LIN {X 0,Y 418.25,Z 362.008,A -85,B 0,C 180,E1 -10239.337,E2 -10239.337} C_VEL
LIN {X 0,Y 418.278,Z 362.011,A -85,B 0,C 180,E1 -10242.396,E2 -10242.396} C_VEL
LIN {X 0,Y 418.299,Z 362.002,A -85,B 0,C 180,E1 -10245.403,E2 -10245.403} C_VEL
LIN {X 0,Y 418.315,Z 361.999,A -85,B 0,C 180,E1 -10248.369,E2 -10248.369} C_VEL
LIN {X 0,Y 418.378,Z 361.987,A -85,B 0,C 180,E1 -10251.305,E2 -10251.305} C_VEL
LIN {X 0,Y 418.49,Z 361.983,A -85,B 0,C 180,E1 -10254.217,E2 -10254.217} C_VEL
LIN {X 0,Y 418.542,Z 361.975,A -85,B 0,C 180,E1 -10258.076,E2 -10258.076} C_VEL
LIN {X 0,Y 418.475,Z 361.982,A -85,B 0,C 180,E1 -10260.963,E2 -10260.963} C_VEL
LIN {X 0,Y 418.488,Z 361.975,A -85,B 0,C 180,E1 -10262.888,E2 -10262.888} C_VEL
LIN {X 0,Y 418.445,Z 361.981,A -85,B 0,C 180,E1 -10266.567,E2 -10266.567} C_VEL
LIN {X 0,Y 418.34,Z 361.998,A -85,B 0,C 180,E1 -10269.672,E2 -10269.672} C_VEL
LIN {X 0,Y 418.349,Z 361.997,A -85,B 0,C 180,E1 -10273.001,E2 -10273.001} C_VEL
LIN {X 0,Y 418.315,Z 362.003,A -85,B 0,C 180,E1 -10276.736,E2 -10276.736} C_VEL
LIN {X 0,Y 418.273,Z 361.985,A -85,B 0,C 180,E1 -10279.79,E2 -10279.79} C_VEL
LIN {X 0,Y 418.233,Z 362.015,A -85,B 0,C 180,E1 -10282.737,E2 -10282.737} C_VEL
LIN {X 0,Y 418.233,Z 361.994,A -85,B 0,C 180,E1 -10285.907,E2 -10285.907} C_VEL
LIN {X 0,Y 418.263,Z 362.006,A -85,B 0,C 180,E1 -10289.163,E2 -10289.163} C_VEL
LIN {X 0,Y 418.26,Z 362.012,A -85,B 0,C 180,E1 -10292.844,E2 -10292.844} C_VEL
LIN {X 0,Y 418.244,Z 362.002,A -85,B 0,C 180,E1 -10296.237,E2 -10296.237} C_VEL
LIN {X 0,Y 418.201,Z 362.009,A -85,B 0,C 180,E1 -10299.688,E2 -10299.688} C_VEL
LIN {X 0,Y 418.215,Z 362.01,A -85,B 0,C 180,E1 -10302.319,E2 -10302.319} C_VEL
LIN {X 0,Y 418.239,Z 362.007,A -85,B 0,C 180,E1 -10305.109,E2 -10305.109} C_VEL
LIN {X 0,Y 418.238,Z 362.008,A -85,B 0,C 180,E1 -10307.766,E2 -10307.766} C_VEL
LIN {X 0,Y 418.259,Z 362.142,A -85,B 0,C 180,E1 -10309.979,E2 -10309.979} C_VEL
LIN {X 0,Y 420.964,Z 372.598,A -85,B 0,C 180,E1 -10312.371,E2 -10312.371} C_VEL
LIN {X 0,Y 430.235,Z 392.629,A -85,B 0,C 180,E1 -10313.476,E2 -10313.476} C_VEL
LIN {X 0,Y 432.008,Z 399.713,A -85,B 0,C 180,E1 -10313.741,E2 -10313.741} C_VEL
LIN {X 0,Y 429.477,Z 524.303,A -85,B 0,C 180,E1 -10315.876,E2 -10315.876} C_VEL
LIN {X 0,Y 429.158,Z 541.846,A -85,B 0,C 180,E1 -10316.252,E2 -10316.252} C_VEL
LIN {X 0,Y 428.401,Z 556.662,A -85,B 0,C 180,E1 -10316.74,E2 -10316.74} C_VEL
LIN {X 0,Y 427.518,Z 571.385,A -85,B 0,C 180,E1 -10317.427,E2 -10317.427} C_VEL
LIN {X 0,Y 426.537,Z 583.995,A -85,B 0,C 180,E1 -10318.179,E2 -10318.179} C_VEL
LIN {X 0,Y 425.351,Z 597.555,A -85,B 0,C 180,E1 -10319.189,E2 -10319.189} C_VEL
LIN {X 0,Y 424.073,Z 610.048,A -85,B 0,C 180,E1 -10320.323,E2 -10320.323} C_VEL
LIN {X 0,Y 422.821,Z 621.605,A -85,B 0,C 180,E1 -10321.586,E2 -10321.586} C_VEL
LIN {X 0,Y 421.617,Z 632.292,A -85,B 0,C 180,E1 -10322.984,E2 -10322.984} C_VEL
LIN {X 0,Y 420.39,Z 642.896,A -85,B 0,C 180,E1 -10324.64,E2 -10324.64} C_VEL
LIN {X 0,Y 419.394,Z 651.646,A -85,B 0,C 180,E1 -10326.285,E2 -10326.285} C_VEL
LIN {X 0,Y 418.644,Z 659.535,A -85,B 0,C 180,E1 -10328.074,E2 -10328.074} C_VEL
LIN {X 0,Y 417.946,Z 665.94,A -85,B 0,C 180,E1 -10329.835,E2 -10329.835} C_VEL
LIN {X 0,Y 417.521,Z 671.781,A -85,B 0,C 180,E1 -10331.856,E2 -10331.856} C_VEL
LIN {X 0,Y 417.395,Z 673.436,A -85,B 0,C 180,E1 -10332.537,E2 -10332.537} C_VEL
LIN {X 0,Y 416.6,Z 675.164,A -85,B 0,C 180,E1 -10333.308,E2 -10333.308} C_VEL
LIN {X 0,Y 413.563,Z 677.628,A -85,B 0,C 180,E1 -10334.568,E2 -10334.568} C_VEL
LIN {X 0,Y 411.054,Z 679.223,A -85,B 0,C 180,E1 -10335.596,E2 -10335.596} C_VEL
LIN {X 0,Y 409.922,Z 680.326,A -85,B 0,C 180,E1 -10336.536,E2 -10336.536} C_VEL
LIN {X 0,Y 409.899,Z 680.381,A -85,B 0,C 180,E1 -10336.673,E2 -10336.673} C_VEL
LIN {X 0,Y 409.94,Z 681.451,A -85,B 0,C 180,E1 -10338.128,E2 -10338.128} C_VEL
LIN {X 0,Y 409.796,Z 681.883,A -85,B 0,C 180,E1 -10340.125,E2 -10340.125} C_VEL
LIN {X 0,Y 409.865,Z 681.164,A -85,B 0,C 180,E1 -10342.116,E2 -10342.116} C_VEL
LIN {X 0,Y 410.059,Z 679.25,A -85,B 0,C 180,E1 -10344.098,E2 -10344.098} C_VEL
LIN {X 0,Y 410.126,Z 676.158,A -85,B 0,C 180,E1 -10346.07,E2 -10346.07} C_VEL
LIN {X 0,Y 410.35,Z 671.836,A -85,B 0,C 180,E1 -10348.037,E2 -10348.037} C_VEL
LIN {X 0,Y 410.68,Z 666.199,A -85,B 0,C 180,E1 -10350,E2 -10350} C_VEL
LIN {X 0,Y 411.345,Z 659.076,A -85,B 0,C 180,E1 -10351.958,E2 -10351.958} C_VEL
LIN {X 0,Y 412.106,Z 651.471,A -85,B 0,C 180,E1 -10353.667,E2 -10353.667} C_VEL
LIN {X 0,Y 413.018,Z 642.359,A -85,B 0,C 180,E1 -10355.37,E2 -10355.37} C_VEL
LIN {X 0,Y 414.008,Z 633.119,A -85,B 0,C 180,E1 -10356.825,E2 -10356.825} C_VEL
LIN {X 0,Y 415.304,Z 621.14,A -85,B 0,C 180,E1 -10358.393,E2 -10358.393} C_VEL
LIN {X 0,Y 416.452,Z 608.984,A -85,B 0,C 180,E1 -10359.716,E2 -10359.716} C_VEL
LIN {X 0,Y 417.684,Z 595.584,A -85,B 0,C 180,E1 -10360.912,E2 -10360.912} C_VEL
LIN {X 0,Y 418.769,Z 582.449,A -85,B 0,C 180,E1 -10361.864,E2 -10361.864} C_VEL
LIN {X 0,Y 419.759,Z 568,A -85,B 0,C 180,E1 -10362.695,E2 -10362.695} C_VEL
LIN {X 0,Y 420.566,Z 552.989,A -85,B 0,C 180,E1 -10363.345,E2 -10363.345} C_VEL
LIN {X 0,Y 421.105,Z 537.257,A -85,B 0,C 180,E1 -10363.82,E2 -10363.82} C_VEL
LIN {X 0,Y 423.525,Z 401.204,A -85,B 0,C 180,E1 -10366.178,E2 -10366.178} C_VEL
LIN {X 0,Y 422.464,Z 395.65,A -85,B 0,C 180,E1 -10366.343,E2 -10366.343} C_VEL
LIN {X 0,Y 421.07,Z 390.956,A -85,B 0,C 180,E1 -10366.513,E2 -10366.513} C_VEL
LIN {X 0,Y 413.404,Z 372.221,A -85,B 0,C 180,E1 -10367.36,E2 -10367.36} C_VEL
LIN {X 0,Y 411.282,Z 362.882,A -85,B 0,C 180,E1 -10369.399,E2 -10369.399} C_VEL
LIN {X 0,Y 411.194,Z 362.89,A -85,B 0,C 180,E1 -10373.148,E2 -10373.148} C_VEL
LIN {X 0,Y 411.18,Z 362.89,A -85,B 0,C 180,E1 -10376.385,E2 -10376.385} C_VEL
LIN {X 0,Y 411.201,Z 362.886,A -85,B 0,C 180,E1 -10379.713,E2 -10379.713} C_VEL
LIN {X 0,Y 411.211,Z 362.881,A -85,B 0,C 180,E1 -10383.156,E2 -10383.156} C_VEL
LIN {X 0,Y 411.193,Z 362.881,A -85,B 0,C 180,E1 -10386.552,E2 -10386.552} C_VEL
LIN {X 0,Y 411.171,Z 362.886,A -85,B 0,C 180,E1 -10389.72,E2 -10389.72} C_VEL
LIN {X 0,Y 411.166,Z 362.892,A -85,B 0,C 180,E1 -10393.135,E2 -10393.135} C_VEL
LIN {X 0,Y 411.169,Z 362.881,A -85,B 0,C 180,E1 -10395.881,E2 -10395.881} C_VEL
LIN {X 0,Y 411.152,Z 362.892,A -85,B 0,C 180,E1 -10398.774,E2 -10398.774} C_VEL
LIN {X 0,Y 411.186,Z 362.89,A -85,B 0,C 180,E1 -10402.025,E2 -10402.025} C_VEL
LIN {X 0,Y 411.206,Z 362.887,A -85,B 0,C 180,E1 -10405.123,E2 -10405.123} C_VEL
LIN {X 0,Y 411.167,Z 362.894,A -85,B 0,C 180,E1 -10408.002,E2 -10408.002} C_VEL
LIN {X 0,Y 411.179,Z 362.878,A -85,B 0,C 180,E1 -10411.406,E2 -10411.406} C_VEL
LIN {X 0,Y 411.191,Z 362.861,A -85,B 0,C 180,E1 -10414.941,E2 -10414.941} C_VEL
LIN {X 0,Y 411.207,Z 362.888,A -85,B 0,C 180,E1 -10417.913,E2 -10417.913} C_VEL
LIN {X 0,Y 411.223,Z 362.883,A -85,B 0,C 180,E1 -10421.051,E2 -10421.051} C_VEL
LIN {X 0,Y 411.257,Z 362.879,A -85,B 0,C 180,E1 -10424.131,E2 -10424.131} C_VEL
LIN {X 0,Y 411.307,Z 362.873,A -85,B 0,C 180,E1 -10427.165,E2 -10427.165} C_VEL
LIN {X 0,Y 411.291,Z 362.873,A -85,B 0,C 180,E1 -10430.161,E2 -10430.161} C_VEL
LIN {X 0,Y 411.393,Z 362.862,A -85,B 0,C 180,E1 -10433.131,E2 -10433.131} C_VEL
LIN {X 0,Y 411.291,Z 362.866,A -85,B 0,C 180,E1 -10435.098,E2 -10435.098} C_VEL
LIN {X 0,Y 411.505,Z 362.849,A -85,B 0,C 180,E1 -10438.042,E2 -10438.042} C_VEL
LIN {X 0,Y 411.517,Z 362.843,A -85,B 0,C 180,E1 -10440,E2 -10440} C_VEL
LIN {X 0,Y 411.449,Z 362.85,A -85,B 0,C 180,E1 -10442.937,E2 -10442.937} C_VEL
LIN {X 0,Y 411.432,Z 362.858,A -85,B 0,C 180,E1 -10445.882,E2 -10445.882} C_VEL
LIN {X 0,Y 411.32,Z 362.866,A -85,B 0,C 180,E1 -10448.846,E2 -10448.846} C_VEL
LIN {X 0,Y 411.285,Z 362.873,A -85,B 0,C 180,E1 -10451.832,E2 -10451.832} C_VEL
LIN {X 0,Y 411.233,Z 362.879,A -85,B 0,C 180,E1 -10454.853,E2 -10454.853} C_VEL
LIN {X 0,Y 411.231,Z 362.878,A -85,B 0,C 180,E1 -10457.916,E2 -10457.916} C_VEL
LIN {X 0,Y 411.198,Z 362.885,A -85,B 0,C 180,E1 -10461.034,E2 -10461.034} C_VEL
LIN {X 0,Y 411.204,Z 362.886,A -85,B 0,C 180,E1 -10464.216,E2 -10464.216} C_VEL
LIN {X 0,Y 411.176,Z 362.891,A -85,B 0,C 180,E1 -10467.483,E2 -10467.483} C_VEL
LIN {X 0,Y 411.197,Z 362.888,A -85,B 0,C 180,E1 -10469.713,E2 -10469.713} C_VEL
LIN {X 0,Y 411.207,Z 362.886,A -85,B 0,C 180,E1 -10473.155,E2 -10473.155} C_VEL
LIN {X 0,Y 411.189,Z 362.887,A -85,B 0,C 180,E1 -10476.551,E2 -10476.551} C_VEL
LIN {X 0,Y 411.167,Z 362.886,A -85,B 0,C 180,E1 -10479.72,E2 -10479.72} C_VEL
LIN {X 0,Y 411.162,Z 362.892,A -85,B 0,C 180,E1 -10483.135,E2 -10483.135} C_VEL
LIN {X 0,Y 411.164,Z 362.895,A -85,B 0,C 180,E1 -10485.881,E2 -10485.881} C_VEL
LIN {X 0,Y 411.148,Z 362.896,A -85,B 0,C 180,E1 -10488.774,E2 -10488.774} C_VEL
LIN {X 0,Y 411.182,Z 362.891,A -85,B 0,C 180,E1 -10492.025,E2 -10492.025} C_VEL
LIN {X 0,Y 411.204,Z 362.891,A -85,B 0,C 180,E1 -10495.666,E2 -10495.666} C_VEL
LIN {X 0,Y 411.212,Z 362.956,A -85,B 0,C 180,E1 -10497.008,E2 -10497.008} C_VEL
LIN {X 0,Y 414.98,Z 378.406,A -85,B 0,C 180,E1 -10500.005,E2 -10500.005} C_VEL
LIN {X 0,Y 417.196,Z 388.376,A -85,B 0,C 180,E1 -10501.856,E2 -10501.856} C_VEL
LIN {X 0,Y 416.892,Z 394.781,A -85,B 0,C 180,E1 -10502.901,E2 -10502.901} C_VEL
LIN {X 0,Y 423.237,Z 429.477,A -85,B 0,C 180,E1 -10503.921,E2 -10503.921} C_VEL
LIN {X 0,Y 420.919,Z 561.659,A -85,B 0,C 180,E1 -10506.213,E2 -10506.213} C_VEL
LIN {X 0,Y 420.155,Z 577.601,A -85,B 0,C 180,E1 -10506.689,E2 -10506.689} C_VEL
LIN {X 0,Y 419.305,Z 592.288,A -85,B 0,C 180,E1 -10507.325,E2 -10507.325} C_VEL
LIN {X 0,Y 418.178,Z 607.066,A -85,B 0,C 180,E1 -10508.171,E2 -10508.171} C_VEL
LIN {X 0,Y 417.022,Z 620.494,A -85,B 0,C 180,E1 -10509.144,E2 -10509.144} C_VEL
LIN {X 0,Y 415.674,Z 634.123,A -85,B 0,C 180,E1 -10510.364,E2 -10510.364} C_VEL
LIN {X 0,Y 414.455,Z 646.627,A -85,B 0,C 180,E1 -10511.732,E2 -10511.732} C_VEL
LIN {X 0,Y 413.378,Z 657.812,A -85,B 0,C 180,E1 -10513.2,E2 -10513.2} C_VEL
LIN {X 0,Y 412.375,Z 667.299,A -85,B 0,C 180,E1 -10514.683,E2 -10514.683} C_VEL
LIN {X 0,Y 411.614,Z 675.377,A -85,B 0,C 180,E1 -10516.17,E2 -10516.17} C_VEL
LIN {X 0,Y 410.988,Z 683.35,A -85,B 0,C 180,E1 -10517.908,E2 -10517.908} C_VEL
LIN {X 0,Y 410.506,Z 689.961,A -85,B 0,C 180,E1 -10519.644,E2 -10519.644} C_VEL
LIN {X 0,Y 410.206,Z 696.028,A -85,B 0,C 180,E1 -10521.626,E2 -10521.626} C_VEL
LIN {X 0,Y 410.056,Z 699.608,A -85,B 0,C 180,E1 -10523.109,E2 -10523.109} C_VEL
LIN {X 0,Y 409.958,Z 703.281,A -85,B 0,C 180,E1 -10525.083,E2 -10525.083} C_VEL
LIN {X 0,Y 409.919,Z 705.726,A -85,B 0,C 180,E1 -10527.052,E2 -10527.052} C_VEL
LIN {X 0,Y 409.935,Z 706.987,A -85,B 0,C 180,E1 -10529.018,E2 -10529.018} C_VEL
LIN {X 0,Y 409.935,Z 707.048,A -85,B 0,C 180,E1 -10530.982,E2 -10530.982} C_VEL
LIN {X 0,Y 409.916,Z 705.971,A -85,B 0,C 180,E1 -10532.948,E2 -10532.948} C_VEL
LIN {X 0,Y 409.94,Z 703.747,A -85,B 0,C 180,E1 -10534.917,E2 -10534.917} C_VEL
LIN {X 0,Y 410.048,Z 700.335,A -85,B 0,C 180,E1 -10536.891,E2 -10536.891} C_VEL
LIN {X 0,Y 410.274,Z 695.646,A -85,B 0,C 180,E1 -10538.869,E2 -10538.869} C_VEL
LIN {X 0,Y 410.686,Z 689.548,A -85,B 0,C 180,E1 -10540.85,E2 -10540.85} C_VEL
LIN {X 0,Y 411.23,Z 682.928,A -85,B 0,C 180,E1 -10542.586,E2 -10542.586} C_VEL
LIN {X 0,Y 412.029,Z 675.001,A -85,B 0,C 180,E1 -10544.319,E2 -10544.319} C_VEL
LIN {X 0,Y 413.047,Z 665.51,A -85,B 0,C 180,E1 -10546.051,E2 -10546.051} C_VEL
LIN {X 0,Y 414.218,Z 655.864,A -85,B 0,C 180,E1 -10547.527,E2 -10547.527} C_VEL
LIN {X 0,Y 415.508,Z 644.448,A -85,B 0,C 180,E1 -10549.002,E2 -10549.002} C_VEL
LIN {X 0,Y 416.82,Z 633.191,A -85,B 0,C 180,E1 -10550.221,E2 -10550.221} C_VEL
LIN {X 0,Y 418.291,Z 619.612,A -85,B 0,C 180,E1 -10551.434,E2 -10551.434} C_VEL
LIN {X 0,Y 419.597,Z 606.311,A -85,B 0,C 180,E1 -10552.399,E2 -10552.399} C_VEL
LIN {X 0,Y 420.822,Z 591.552,A -85,B 0,C 180,E1 -10553.246,E2 -10553.246} C_VEL
LIN {X 0,Y 421.861,Z 576.455,A -85,B 0,C 180,E1 -10553.893,E2 -10553.893} C_VEL
LIN {X 0,Y 422.653,Z 561.479,A -85,B 0,C 180,E1 -10554.335,E2 -10554.335} C_VEL
LIN {X 0,Y 424.423,Z 477.264,A -85,B 0,C 180,E1 -10555.827,E2 -10555.827} C_VEL
LIN {X 0,Y 425.245,Z 428.739,A -85,B 0,C 180,E1 -10556.686,E2 -10556.686} C_VEL
LIN {X 0,Y 420.958,Z 406.331,A -85,B 0,C 180,E1 -10557.445,E2 -10557.445} C_VEL
LIN {X 0,Y 418.176,Z 394.198,A -85,B 0,C 180,E1 -10557.913,E2 -10557.913} C_VEL
LIN {X 0,Y 418.264,Z 390.82,A -85,B 0,C 180,E1 -10558.508,E2 -10558.508} C_VEL
LIN {X 0,Y 415.766,Z 379.592,A -85,B 0,C 180,E1 -10560.752,E2 -10560.752} C_VEL
LIN {X 0,Y 411.97,Z 365.752,A -85,B 0,C 180,E1 -10563.716,E2 -10563.716} C_VEL
LIN {X 0,Y 411.242,Z 362.886,A -85,B 0,C 180,E1 -10564.398,E2 -10564.398} C_VEL
LIN {X 0,Y 411.191,Z 362.888,A -85,B 0,C 180,E1 -10568.166,E2 -10568.166} C_VEL
LIN {X 0,Y 411.162,Z 362.885,A -85,B 0,C 180,E1 -10571.807,E2 -10571.807} C_VEL
LIN {X 0,Y 411.173,Z 362.892,A -85,B 0,C 180,E1 -10575.51,E2 -10575.51} C_VEL
LIN {X 0,Y 411.146,Z 362.897,A -85,B 0,C 180,E1 -10578.775,E2 -10578.775} C_VEL
LIN {X 0,Y 411.181,Z 362.892,A -85,B 0,C 180,E1 -10582.025,E2 -10582.025} C_VEL
LIN {X 0,Y 411.205,Z 362.883,A -85,B 0,C 180,E1 -10585.667,E2 -10585.667} C_VEL
LIN {X 0,Y 411.188,Z 362.868,A -85,B 0,C 180,E1 -10589.153,E2 -10589.153} C_VEL
LIN {X 0,Y 411.188,Z 362.89,A -85,B 0,C 180,E1 -10592.518,E2 -10592.518} C_VEL
LIN {X 0,Y 411.211,Z 362.886,A -85,B 0,C 180,E1 -10595.784,E2 -10595.784} C_VEL
LIN {X 0,Y 411.197,Z 362.888,A -85,B 0,C 180,E1 -10598.966,E2 -10598.966} C_VEL
LIN {X 0,Y 411.244,Z 362.883,A -85,B 0,C 180,E1 -10602.085,E2 -10602.085} C_VEL
LIN {X 0,Y 411.256,Z 362.88,A -85,B 0,C 180,E1 -10605.148,E2 -10605.148} C_VEL
LIN {X 0,Y 411.284,Z 362.873,A -85,B 0,C 180,E1 -10608.168,E2 -10608.168} C_VEL
LIN {X 0,Y 411.319,Z 362.867,A -85,B 0,C 180,E1 -10611.154,E2 -10611.154} C_VEL
LIN {X 0,Y 411.435,Z 362.861,A -85,B 0,C 180,E1 -10614.118,E2 -10614.118} C_VEL
LIN {X 0,Y 411.511,Z 362.851,A -85,B 0,C 180,E1 -10618.043,E2 -10618.043} C_VEL
LIN {X 0,Y 411.439,Z 362.859,A -85,B 0,C 180,E1 -10620.979,E2 -10620.979} C_VEL
LIN {X 0,Y 411.445,Z 362.851,A -85,B 0,C 180,E1 -10622.938,E2 -10622.938} C_VEL
LIN {X 0,Y 411.394,Z 362.858,A -85,B 0,C 180,E1 -10626.564,E2 -10626.564} C_VEL
LIN {X 0,Y 411.292,Z 362.876,A -85,B 0,C 180,E1 -10629.839,E2 -10629.839} C_VEL
LIN {X 0,Y 411.308,Z 362.874,A -85,B 0,C 180,E1 -10633.105,E2 -10633.105} C_VEL
LIN {X 0,Y 411.26,Z 362.88,A -85,B 0,C 180,E1 -10636.889,E2 -10636.889} C_VEL
LIN {X 0,Y 411.233,Z 362.862,A -85,B 0,C 180,E1 -10639.987,E2 -10639.987} C_VEL
LIN {X 0,Y 411.195,Z 362.888,A -85,B 0,C 180,E1 -10643.149,E2 -10643.149} C_VEL
LIN {X 0,Y 411.202,Z 362.872,A -85,B 0,C 180,E1 -10646.384,E2 -10646.384} C_VEL
LIN {X 0,Y 411.201,Z 362.885,A -85,B 0,C 180,E1 -10649.713,E2 -10649.713} C_VEL
LIN {X 0,Y 411.209,Z 362.888,A -85,B 0,C 180,E1 -10653.156,E2 -10653.156} C_VEL
LIN {X 0,Y 411.193,Z 362.884,A -85,B 0,C 180,E1 -10656.552,E2 -10656.552} C_VEL
LIN {X 0,Y 411.171,Z 362.884,A -85,B 0,C 180,E1 -10659.72,E2 -10659.72} C_VEL
LIN {X 0,Y 411.168,Z 362.89,A -85,B 0,C 180,E1 -10663.135,E2 -10663.135} C_VEL
LIN {X 0,Y 411.171,Z 362.889,A -85,B 0,C 180,E1 -10665.881,E2 -10665.881} C_VEL
LIN {X 0,Y 411.202,Z 362.968,A -85,B 0,C 180,E1 -10669.463,E2 -10669.463} C_VEL
LIN {X 0,Y 413.805,Z 372.82,A -85,B 0,C 180,E1 -10671.785,E2 -10671.785} C_VEL
LIN {X 0,Y 423.326,Z 393.023,A -85,B 0,C 180,E1 -10672.955,E2 -10672.955} C_VEL
LIN {X 0,Y 425.12,Z 397.783,A -85,B 0,C 180,E1 -10673.186,E2 -10673.186} C_VEL
LIN {X 0,Y 425.799,Z 401.91,A -85,B 0,C 180,E1 -10673.317,E2 -10673.317} C_VEL
LIN {X 0,Y 423.16,Z 524.186,A -85,B 0,C 180,E1 -10675.439,E2 -10675.439} C_VEL
LIN {X 0,Y 422.809,Z 542.115,A -85,B 0,C 180,E1 -10675.828,E2 -10675.828} C_VEL
LIN {X 0,Y 422,Z 557.264,A -85,B 0,C 180,E1 -10676.336,E2 -10676.336} C_VEL
LIN {X 0,Y 421.104,Z 571.48,A -85,B 0,C 180,E1 -10677.01,E2 -10677.01} C_VEL
LIN {X 0,Y 420.077,Z 584.11,A -85,B 0,C 180,E1 -10677.773,E2 -10677.773} C_VEL
LIN {X 0,Y 418.863,Z 597.388,A -85,B 0,C 180,E1 -10678.771,E2 -10678.771} C_VEL
LIN {X 0,Y 417.486,Z 610.188,A -85,B 0,C 180,E1 -10679.946,E2 -10679.946} C_VEL
LIN {X 0,Y 416.212,Z 621.333,A -85,B 0,C 180,E1 -10681.179,E2 -10681.179} C_VEL
LIN {X 0,Y 414.785,Z 633.349,A -85,B 0,C 180,E1 -10682.775,E2 -10682.775} C_VEL
LIN {X 0,Y 413.627,Z 642.479,A -85,B 0,C 180,E1 -10684.23,E2 -10684.23} C_VEL
LIN {X 0,Y 412.606,Z 651.177,A -85,B 0,C 180,E1 -10685.871,E2 -10685.871} C_VEL
LIN {X 0,Y 411.809,Z 658.532,A -85,B 0,C 180,E1 -10687.523,E2 -10687.523} C_VEL
LIN {X 0,Y 410.999,Z 665.706,A -85,B 0,C 180,E1 -10689.479,E2 -10689.479} C_VEL
LIN {X 0,Y 410.524,Z 671.653,A -85,B 0,C 180,E1 -10691.536,E2 -10691.536} C_VEL
LIN {X 0,Y 410.213,Z 676.214,A -85,B 0,C 180,E1 -10693.624,E2 -10693.624} C_VEL
LIN {X 0,Y 409.996,Z 678.604,A -85,B 0,C 180,E1 -10695.101,E2 -10695.101} C_VEL
LIN {X 0,Y 409.899,Z 680.381,A -85,B 0,C 180,E1 -10696.673,E2 -10696.673} C_VEL
LIN {X 0,Y 409.226,Z 681.121,A -85,B 0,C 180,E1 -10697.487,E2 -10697.487} C_VEL
LIN {X 0,Y 406.332,Z 681.935,A -85,B 0,C 180,E1 -10698.815,E2 -10698.815} C_VEL
LIN {X 0,Y 403.881,Z 682.179,A -85,B 0,C 180,E1 -10699.889,E2 -10699.889} C_VEL
LIN {X 0,Y 402.824,Z 682.045,A -85,B 0,C 180,E1 -10700.72,E2 -10700.72} C_VEL
LIN {X 0,Y 402.736,Z 681.93,A -85,B 0,C 180,E1 -10701.002,E2 -10701.002} C_VEL
LIN {X 0,Y 402.865,Z 680.687,A -85,B 0,C 180,E1 -10702.986,E2 -10702.986} C_VEL
LIN {X 0,Y 402.98,Z 678.269,A -85,B 0,C 180,E1 -10704.997,E2 -10704.997} C_VEL
LIN {X 0,Y 403.218,Z 674.655,A -85,B 0,C 180,E1 -10707.003,E2 -10707.003} C_VEL
LIN {X 0,Y 403.369,Z 669.795,A -85,B 0,C 180,E1 -10709.002,E2 -10709.002} C_VEL
LIN {X 0,Y 403.926,Z 663.534,A -85,B 0,C 180,E1 -10710.997,E2 -10710.997} C_VEL
LIN {X 0,Y 404.734,Z 655.704,A -85,B 0,C 180,E1 -10712.986,E2 -10712.986} C_VEL
LIN {X 0,Y 405.593,Z 647.389,A -85,B 0,C 180,E1 -10714.721,E2 -10714.721} C_VEL
LIN {X 0,Y 406.658,Z 637.404,A -85,B 0,C 180,E1 -10716.45,E2 -10716.45} C_VEL
LIN {X 0,Y 407.786,Z 627.23,A -85,B 0,C 180,E1 -10717.925,E2 -10717.925} C_VEL
LIN {X 0,Y 409.129,Z 615.05,A -85,B 0,C 180,E1 -10719.392,E2 -10719.392} C_VEL
LIN {X 0,Y 410.27,Z 602.923,A -85,B 0,C 180,E1 -10720.612,E2 -10720.612} C_VEL
LIN {X 0,Y 411.554,Z 589.652,A -85,B 0,C 180,E1 -10721.7,E2 -10721.7} C_VEL
LIN {X 0,Y 412.651,Z 574.974,A -85,B 0,C 180,E1 -10722.667,E2 -10722.667} C_VEL
LIN {X 0,Y 413.58,Z 560.736,A -85,B 0,C 180,E1 -10723.387,E2 -10723.387} C_VEL
LIN {X 0,Y 414.27,Z 545.396,A -85,B 0,C 180,E1 -10723.959,E2 -10723.959} C_VEL
LIN {X 0,Y 414.753,Z 530.394,A -85,B 0,C 180,E1 -10724.317,E2 -10724.317} C_VEL
LIN {X 0,Y 417.023,Z 401.358,A -85,B 0,C 180,E1 -10726.569,E2 -10726.569} C_VEL
LIN {X 0,Y 415.255,Z 394.549,A -85,B 0,C 180,E1 -10726.805,E2 -10726.805} C_VEL
LIN {X 0,Y 406.209,Z 372.398,A -85,B 0,C 180,E1 -10727.836,E2 -10727.836} C_VEL
LIN {X 0,Y 404.2,Z 363.763,A -85,B 0,C 180,E1 -10729.739,E2 -10729.739} C_VEL
LIN {X 0,Y 404.154,Z 363.768,A -85,B 0,C 180,E1 -10733.576,E2 -10733.576} C_VEL
LIN {X 0,Y 404.123,Z 363.77,A -85,B 0,C 180,E1 -10736.882,E2 -10736.882} C_VEL
LIN {X 0,Y 404.148,Z 363.765,A -85,B 0,C 180,E1 -10740.285,E2 -10740.285} C_VEL
LIN {X 0,Y 404.149,Z 363.769,A -85,B 0,C 180,E1 -10743.812,E2 -10743.812} C_VEL
LIN {X 0,Y 404.135,Z 363.761,A -85,B 0,C 180,E1 -10746.874,E2 -10746.874} C_VEL
LIN {X 0,Y 404.12,Z 363.761,A -85,B 0,C 180,E1 -10750.074,E2 -10750.074} C_VEL
LIN {X 0,Y 404.146,Z 363.767,A -85,B 0,C 180,E1 -10753.082,E2 -10753.082} C_VEL
LIN {X 0,Y 404.149,Z 363.755,A -85,B 0,C 180,E1 -10755.925,E2 -10755.925} C_VEL
LIN {X 0,Y 404.107,Z 363.77,A -85,B 0,C 180,E1 -10758.633,E2 -10758.633} C_VEL
LIN {X 0,Y 404.141,Z 363.765,A -85,B 0,C 180,E1 -10761.495,E2 -10761.495} C_VEL
LIN {X 0,Y 404.177,Z 363.762,A -85,B 0,C 180,E1 -10764.982,E2 -10764.982} C_VEL
LIN {X 0,Y 404.142,Z 363.767,A -85,B 0,C 180,E1 -10768.442,E2 -10768.442} C_VEL
LIN {X 0,Y 404.155,Z 363.76,A -85,B 0,C 180,E1 -10770.862,E2 -10770.862} C_VEL
LIN {X 0,Y 404.155,Z 363.736,A -85,B 0,C 180,E1 -10774.722,E2 -10774.722} C_VEL
LIN {X 0,Y 404.17,Z 363.759,A -85,B 0,C 180,E1 -10777.508,E2 -10777.508} C_VEL
LIN {X 0,Y 404.166,Z 363.761,A -85,B 0,C 180,E1 -10780.707,E2 -10780.707} C_VEL
LIN {X 0,Y 404.224,Z 363.756,A -85,B 0,C 180,E1 -10783.848,E2 -10783.848} C_VEL
LIN {X 0,Y 404.286,Z 363.746,A -85,B 0,C 180,E1 -10786.938,E2 -10786.938} C_VEL
LIN {X 0,Y 404.257,Z 363.75,A -85,B 0,C 180,E1 -10789.988,E2 -10789.988} C_VEL
LIN {X 0,Y 404.343,Z 363.739,A -85,B 0,C 180,E1 -10793.011,E2 -10793.011} C_VEL
LIN {X 0,Y 404.262,Z 363.741,A -85,B 0,C 180,E1 -10795.013,E2 -10795.013} C_VEL
LIN {X 0,Y 404.474,Z 363.726,A -85,B 0,C 180,E1 -10798.008,E2 -10798.008} C_VEL
LIN {X 0,Y 404.353,Z 363.733,A -85,B 0,C 180,E1 -10800.995,E2 -10800.995} C_VEL
LIN {X 0,Y 404.407,Z 363.727,A -85,B 0,C 180,E1 -10802.988,E2 -10802.988} C_VEL
LIN {X 0,Y 404.38,Z 363.735,A -85,B 0,C 180,E1 -10805.985,E2 -10805.985} C_VEL
LIN {X 0,Y 404.267,Z 363.746,A -85,B 0,C 180,E1 -10809.001,E2 -10809.001} C_VEL
LIN {X 0,Y 404.258,Z 363.746,A -85,B 0,C 180,E1 -10812.041,E2 -10812.041} C_VEL
LIN {X 0,Y 404.178,Z 363.759,A -85,B 0,C 180,E1 -10815.119,E2 -10815.119} C_VEL
LIN {X 0,Y 404.195,Z 363.754,A -85,B 0,C 180,E1 -10818.238,E2 -10818.238} C_VEL
LIN {X 0,Y 404.16,Z 363.764,A -85,B 0,C 180,E1 -10821.418,E2 -10821.418} C_VEL
LIN {X 0,Y 404.161,Z 363.762,A -85,B 0,C 180,E1 -10824.666,E2 -10824.666} C_VEL
LIN {X 0,Y 404.119,Z 363.771,A -85,B 0,C 180,E1 -10828.005,E2 -10828.005} C_VEL
LIN {X 0,Y 404.144,Z 363.765,A -85,B 0,C 180,E1 -10830.285,E2 -10830.285} C_VEL
LIN {X 0,Y 404.145,Z 363.77,A -85,B 0,C 180,E1 -10833.812,E2 -10833.812} C_VEL
LIN {X 0,Y 404.131,Z 363.767,A -85,B 0,C 180,E1 -10836.874,E2 -10836.874} C_VEL
LIN {X 0,Y 404.116,Z 363.766,A -85,B 0,C 180,E1 -10840.074,E2 -10840.074} C_VEL
LIN {X 0,Y 404.141,Z 363.766,A -85,B 0,C 180,E1 -10843.082,E2 -10843.082} C_VEL
LIN {X 0,Y 404.144,Z 363.77,A -85,B 0,C 180,E1 -10845.925,E2 -10845.925} C_VEL
LIN {X 0,Y 404.103,Z 363.773,A -85,B 0,C 180,E1 -10848.633,E2 -10848.633} C_VEL
LIN {X 0,Y 404.137,Z 363.771,A -85,B 0,C 180,E1 -10851.495,E2 -10851.495} C_VEL
LIN {X 0,Y 404.182,Z 363.764,A -85,B 0,C 180,E1 -10854.983,E2 -10854.983} C_VEL
LIN {X 0,Y 404.152,Z 363.787,A -85,B 0,C 180,E1 -10856.622,E2 -10856.622} C_VEL
LIN {X 0,Y 408.039,Z 379.537,A -85,B 0,C 180,E1 -10859.742,E2 -10859.742} C_VEL
LIN {X 0,Y 410.222,Z 389.419,A -85,B 0,C 180,E1 -10861.613,E2 -10861.613} C_VEL
LIN {X 0,Y 410.299,Z 392.644,A -85,B 0,C 180,E1 -10862.175,E2 -10862.175} C_VEL
LIN {X 0,Y 410.093,Z 394.337,A -85,B 0,C 180,E1 -10862.455,E2 -10862.455} C_VEL
LIN {X 0,Y 416.719,Z 430.136,A -85,B 0,C 180,E1 -10863.546,E2 -10863.546} C_VEL
LIN {X 0,Y 414.323,Z 560.95,A -85,B 0,C 180,E1 -10865.844,E2 -10865.844} C_VEL
LIN {X 0,Y 413.519,Z 577.111,A -85,B 0,C 180,E1 -10866.327,E2 -10866.327} C_VEL
LIN {X 0,Y 412.693,Z 591.244,A -85,B 0,C 180,E1 -10866.941,E2 -10866.941} C_VEL
LIN {X 0,Y 411.538,Z 606.224,A -85,B 0,C 180,E1 -10867.8,E2 -10867.8} C_VEL
LIN {X 0,Y 410.309,Z 619.75,A -85,B 0,C 180,E1 -10868.787,E2 -10868.787} C_VEL
LIN {X 0,Y 408.892,Z 633.495,A -85,B 0,C 180,E1 -10870.025,E2 -10870.025} C_VEL
LIN {X 0,Y 407.74,Z 645.223,A -85,B 0,C 180,E1 -10871.314,E2 -10871.314} C_VEL
LIN {X 0,Y 406.475,Z 657.309,A -85,B 0,C 180,E1 -10872.906,E2 -10872.906} C_VEL
LIN {X 0,Y 405.302,Z 668.308,A -85,B 0,C 180,E1 -10874.666,E2 -10874.666} C_VEL
LIN {X 0,Y 404.396,Z 677.675,A -85,B 0,C 180,E1 -10876.482,E2 -10876.482} C_VEL
LIN {X 0,Y 403.758,Z 685.995,A -85,B 0,C 180,E1 -10878.453,E2 -10878.453} C_VEL
LIN {X 0,Y 403.236,Z 692.848,A -85,B 0,C 180,E1 -10880.469,E2 -10880.469} C_VEL
LIN {X 0,Y 403.026,Z 698.223,A -85,B 0,C 180,E1 -10882.485,E2 -10882.485} C_VEL
LIN {X 0,Y 402.896,Z 701.316,A -85,B 0,C 180,E1 -10883.992,E2 -10883.992} C_VEL
LIN {X 0,Y 402.826,Z 704.392,A -85,B 0,C 180,E1 -10885.998,E2 -10885.998} C_VEL
LIN {X 0,Y 402.902,Z 706.272,A -85,B 0,C 180,E1 -10888.001,E2 -10888.001} C_VEL
LIN {X 0,Y 402.848,Z 706.935,A -85,B 0,C 180,E1 -10890,E2 -10890} C_VEL
LIN {X 0,Y 402.886,Z 706.451,A -85,B 0,C 180,E1 -10891.999,E2 -10891.999} C_VEL
LIN {X 0,Y 402.821,Z 704.826,A -85,B 0,C 180,E1 -10894.002,E2 -10894.002} C_VEL
LIN {X 0,Y 402.896,Z 701.825,A -85,B 0,C 180,E1 -10896.127,E2 -10896.127} C_VEL
LIN {X 0,Y 403.066,Z 698.03,A -85,B 0,C 180,E1 -10898.018,E2 -10898.018} C_VEL
LIN {X 0,Y 403.348,Z 692.669,A -85,B 0,C 180,E1 -10900.034,E2 -10900.034} C_VEL
LIN {X 0,Y 404.02,Z 685.857,A -85,B 0,C 180,E1 -10902.049,E2 -10902.049} C_VEL
LIN {X 0,Y 404.655,Z 678.652,A -85,B 0,C 180,E1 -10903.791,E2 -10903.791} C_VEL
LIN {X 0,Y 405.655,Z 669.795,A -85,B 0,C 180,E1 -10905.577,E2 -10905.577} C_VEL
LIN {X 0,Y 406.948,Z 659.307,A -85,B 0,C 180,E1 -10907.332,E2 -10907.332} C_VEL
LIN {X 0,Y 408.387,Z 647.909,A -85,B 0,C 180,E1 -10908.914,E2 -10908.914} C_VEL
LIN {X 0,Y 409.863,Z 635.736,A -85,B 0,C 180,E1 -10910.318,E2 -10910.318} C_VEL
LIN {X 0,Y 411.344,Z 622.778,A -85,B 0,C 180,E1 -10911.552,E2 -10911.552} C_VEL
LIN {X 0,Y 412.907,Z 608.473,A -85,B 0,C 180,E1 -10912.65,E2 -10912.65} C_VEL
LIN {X 0,Y 414.175,Z 593.896,A -85,B 0,C 180,E1 -10913.538,E2 -10913.538} C_VEL
LIN {X 0,Y 415.302,Z 578.854,A -85,B 0,C 180,E1 -10914.228,E2 -10914.228} C_VEL
LIN {X 0,Y 416.216,Z 564.026,A -85,B 0,C 180,E1 -10914.703,E2 -10914.703} C_VEL
LIN {X 0,Y 416.802,Z 544.454,A -85,B 0,C 180,E1 -10915.099,E2 -10915.099} C_VEL
LIN {X 0,Y 419.05,Z 429.9,A -85,B 0,C 180,E1 -10917.137,E2 -10917.137} C_VEL
LIN {X 0,Y 414.651,Z 406.882,A -85,B 0,C 180,E1 -10917.938,E2 -10917.938} C_VEL
LIN {X 0,Y 411.647,Z 393.931,A -85,B 0,C 180,E1 -10918.461,E2 -10918.461} C_VEL
LIN {X 0,Y 409.506,Z 383.486,A -85,B 0,C 180,E1 -10920.563,E2 -10920.563} C_VEL
LIN {X 0,Y 405.965,Z 370.221,A -85,B 0,C 180,E1 -10923.43,E2 -10923.43} C_VEL
LIN {X 0,Y 404.163,Z 363.767,A -85,B 0,C 180,E1 -10924.942,E2 -10924.942} C_VEL
LIN {X 0,Y 404.137,Z 363.762,A -85,B 0,C 180,E1 -10928.505,E2 -10928.505} C_VEL
LIN {X 0,Y 404.107,Z 363.764,A -85,B 0,C 180,E1 -10931.598,E2 -10931.598} C_VEL
LIN {X 0,Y 404.143,Z 363.768,A -85,B 0,C 180,E1 -10934.522,E2 -10934.522} C_VEL
LIN {X 0,Y 404.121,Z 363.77,A -85,B 0,C 180,E1 -10937.294,E2 -10937.294} C_VEL
LIN {X 0,Y 404.131,Z 363.77,A -85,B 0,C 180,E1 -10939.951,E2 -10939.951} C_VEL
LIN {X 0,Y 404.131,Z 363.756,A -85,B 0,C 180,E1 -10943.126,E2 -10943.126} C_VEL
LIN {X 0,Y 404.144,Z 363.767,A -85,B 0,C 180,E1 -10946.188,E2 -10946.188} C_VEL
LIN {X 0,Y 404.144,Z 363.747,A -85,B 0,C 180,E1 -10949.715,E2 -10949.715} C_VEL
LIN {X 0,Y 404.134,Z 363.763,A -85,B 0,C 180,E1 -10953.119,E2 -10953.119} C_VEL
LIN {X 0,Y 404.16,Z 363.764,A -85,B 0,C 180,E1 -10956.425,E2 -10956.425} C_VEL
LIN {X 0,Y 404.192,Z 363.761,A -85,B 0,C 180,E1 -10959.875,E2 -10959.875} C_VEL
LIN {X 0,Y 404.216,Z 363.755,A -85,B 0,C 180,E1 -10962.994,E2 -10962.994} C_VEL
LIN {X 0,Y 404.284,Z 363.746,A -85,B 0,C 180,E1 -10966.939,E2 -10966.939} C_VEL
LIN {X 0,Y 404.257,Z 363.754,A -85,B 0,C 180,E1 -10969.989,E2 -10969.989} C_VEL
LIN {X 0,Y 404.344,Z 363.742,A -85,B 0,C 180,E1 -10973.012,E2 -10973.012} C_VEL
LIN {X 0,Y 404.271,Z 363.745,A -85,B 0,C 180,E1 -10975.014,E2 -10975.014} C_VEL
LIN {X 0,Y 404.479,Z 363.726,A -85,B 0,C 180,E1 -10978.009,E2 -10978.009} C_VEL
LIN {X 0,Y 404.404,Z 363.735,A -85,B 0,C 180,E1 -10980.996,E2 -10980.996} C_VEL
LIN {X 0,Y 404.403,Z 363.728,A -85,B 0,C 180,E1 -10982.989,E2 -10982.989} C_VEL
LIN {X 0,Y 404.346,Z 363.737,A -85,B 0,C 180,E1 -10986.56,E2 -10986.56} C_VEL
LIN {X 0,Y 404.267,Z 363.752,A -85,B 0,C 180,E1 -10989.002,E2 -10989.002} C_VEL
LIN {X 0,Y 404.258,Z 363.75,A -85,B 0,C 180,E1 -10992.042,E2 -10992.042} C_VEL
LIN {X 0,Y 404.208,Z 363.757,A -85,B 0,C 180,E1 -10995.118,E2 -10995.118} C_VEL
LIN {X 0,Y 404.211,Z 363.749,A -85,B 0,C 180,E1 -10998.239,E2 -10998.239} C_VEL
LIN {X 0,Y 404.141,Z 363.762,A -85,B 0,C 180,E1 -11001.42,E2 -11001.42} C_VEL
LIN {X 0,Y 404.153,Z 363.753,A -85,B 0,C 180,E1 -11004.668,E2 -11004.668} C_VEL
LIN {X 0,Y 404.169,Z 363.762,A -85,B 0,C 180,E1 -11008.002,E2 -11008.002} C_VEL
LIN {X 0,Y 404.142,Z 363.756,A -85,B 0,C 180,E1 -11011.558,E2 -11011.558} C_VEL
LIN {X 0,Y 404.181,Z 363.75,A -85,B 0,C 180,E1 -11015.017,E2 -11015.017} C_VEL
LIN {X 0,Y 404.135,Z 363.761,A -85,B 0,C 180,E1 -11018.76,E2 -11018.76} C_VEL
LIN {X 0,Y 404.111,Z 363.771,A -85,B 0,C 180,E1 -11021.598,E2 -11021.598} C_VEL
LIN {X 0,Y 404.147,Z 363.767,A -85,B 0,C 180,E1 -11024.522,E2 -11024.522} C_VEL
LIN {X 0,Y 404.136,Z 363.766,A -85,B 0,C 180,E1 -11027.295,E2 -11027.295} C_VEL
LIN {X 0,Y 404.144,Z 363.796,A -85,B 0,C 180,E1 -11028.926,E2 -11028.926} C_VEL
LIN {X 0,Y 406.713,Z 373.268,A -85,B 0,C 180,E1 -11031.183,E2 -11031.183} C_VEL
LIN {X 0,Y 416.804,Z 394.292,A -85,B 0,C 180,E1 -11032.46,E2 -11032.46} C_VEL
LIN {X 0,Y 419.145,Z 399.967,A -85,B 0,C 180,E1 -11032.759,E2 -11032.759} C_VEL
LIN {X 0,Y 419.646,Z 402.366,A -85,B 0,C 180,E1 -11032.846,E2 -11032.846} C_VEL
LIN {X 0,Y 416.869,Z 524.178,A -85,B 0,C 180,E1 -11034.989,E2 -11034.989} C_VEL
LIN {X 0,Y 416.516,Z 541.374,A -85,B 0,C 180,E1 -11035.36,E2 -11035.36} C_VEL
LIN {X 0,Y 415.72,Z 556.51,A -85,B 0,C 180,E1 -11035.864,E2 -11035.864} C_VEL
LIN {X 0,Y 414.714,Z 571.61,A -85,B 0,C 180,E1 -11036.58,E2 -11036.58} C_VEL
LIN {X 0,Y 413.636,Z 584.253,A -85,B 0,C 180,E1 -11037.353,E2 -11037.353} C_VEL
LIN {X 0,Y 412.335,Z 597.849,A -85,B 0,C 180,E1 -11038.393,E2 -11038.393} C_VEL
LIN {X 0,Y 410.922,Z 610.349,A -85,B 0,C 180,E1 -11039.557,E2 -11039.557} C_VEL
LIN {X 0,Y 409.51,Z 622.038,A -85,B 0,C 180,E1 -11040.873,E2 -11040.873} C_VEL
LIN {X 0,Y 407.933,Z 634.361,A -85,B 0,C 180,E1 -11042.558,E2 -11042.558} C_VEL
LIN {X 0,Y 406.711,Z 643.712,A -85,B 0,C 180,E1 -11044.088,E2 -11044.088} C_VEL
LIN {X 0,Y 405.524,Z 653.24,A -85,B 0,C 180,E1 -11045.967,E2 -11045.967} C_VEL
LIN {X 0,Y 404.769,Z 659.858,A -85,B 0,C 180,E1 -11047.543,E2 -11047.543} C_VEL
LIN {X 0,Y 403.895,Z 667.132,A -85,B 0,C 180,E1 -11049.634,E2 -11049.634} C_VEL
LIN {X 0,Y 403.423,Z 672.796,A -85,B 0,C 180,E1 -11051.725,E2 -11051.725} C_VEL
LIN {X 0,Y 403.121,Z 677.013,A -85,B 0,C 180,E1 -11053.803,E2 -11053.803} C_VEL
LIN {X 0,Y 402.853,Z 679.921,A -85,B 0,C 180,E1 -11055.863,E2 -11055.863} C_VEL
LIN {X 0,Y 402.862,Z 681.605,A -85,B 0,C 180,E1 -11057.916,E2 -11057.916} C_VEL
LIN {X 0,Y 402.715,Z 682.125,A -85,B 0,C 180,E1 -11059.95,E2 -11059.95} C_VEL
LIN {X 0,Y 402.736,Z 681.93,A -85,B 0,C 180,E1 -11061.002,E2 -11061.002} C_VEL
LIN {X 0,Y 402.078,Z 681.561,A -85,B 0,C 180,E1 -11061.836,E2 -11061.836} C_VEL
LIN {X 0,Y 399.288,Z 680.633,A -85,B 0,C 180,E1 -11063.191,E2 -11063.191} C_VEL
LIN {X 0,Y 396.947,Z 679.518,A -85,B 0,C 180,E1 -11064.28,E2 -11064.28} C_VEL
LIN {X 0,Y 395.964,Z 678.388,A -85,B 0,C 180,E1 -11065.113,E2 -11065.113} C_VEL
LIN {X 0,Y 395.896,Z 677.918,A -85,B 0,C 180,E1 -11065.393,E2 -11065.393} C_VEL
LIN {X 0,Y 396.146,Z 674.102,A -85,B 0,C 180,E1 -11067.458,E2 -11067.458} C_VEL
LIN {X 0,Y 396.399,Z 668.98,A -85,B 0,C 180,E1 -11069.492,E2 -11069.492} C_VEL
LIN {X 0,Y 397.063,Z 662.438,A -85,B 0,C 180,E1 -11071.521,E2 -11071.521} C_VEL
LIN {X 0,Y 397.807,Z 655.403,A -85,B 0,C 180,E1 -11073.292,E2 -11073.292} C_VEL
LIN {X 0,Y 398.713,Z 646.977,A -85,B 0,C 180,E1 -11075.056,E2 -11075.056} C_VEL
LIN {X 0,Y 399.853,Z 636.863,A -85,B 0,C 180,E1 -11076.814,E2 -11076.814} C_VEL
LIN {X 0,Y 401.07,Z 626.529,A -85,B 0,C 180,E1 -11078.312,E2 -11078.312} C_VEL
LIN {X 0,Y 402.341,Z 615.317,A -85,B 0,C 180,E1 -11079.679,E2 -11079.679} C_VEL
LIN {X 0,Y 403.513,Z 603.194,A -85,B 0,C 180,E1 -11080.918,E2 -11080.918} C_VEL
LIN {X 0,Y 404.841,Z 589.93,A -85,B 0,C 180,E1 -11082.024,E2 -11082.024} C_VEL
LIN {X 0,Y 405.982,Z 575.27,A -85,B 0,C 180,E1 -11083.006,E2 -11083.006} C_VEL
LIN {X 0,Y 406.953,Z 561.04,A -85,B 0,C 180,E1 -11083.737,E2 -11083.737} C_VEL
LIN {X 0,Y 407.679,Z 545.726,A -85,B 0,C 180,E1 -11084.316,E2 -11084.316} C_VEL
LIN {X 0,Y 408.175,Z 530.791,A -85,B 0,C 180,E1 -11084.681,E2 -11084.681} C_VEL
LIN {X 0,Y 410.55,Z 403.013,A -85,B 0,C 180,E1 -11086.942,E2 -11086.942} C_VEL
LIN {X 0,Y 409.059,Z 396.947,A -85,B 0,C 180,E1 -11087.152,E2 -11087.152} C_VEL
LIN {X 0,Y 399.053,Z 372.704,A -85,B 0,C 180,E1 -11088.298,E2 -11088.298} C_VEL
LIN {X 0,Y 397.158,Z 364.634,A -85,B 0,C 180,E1 -11090.129,E2 -11090.129} C_VEL
LIN {X 0,Y 397.117,Z 364.644,A -85,B 0,C 180,E1 -11094.019,E2 -11094.019} C_VEL
LIN {X 0,Y 397.084,Z 364.649,A -85,B 0,C 180,E1 -11097.753,E2 -11097.753} C_VEL
LIN {X 0,Y 397.082,Z 364.645,A -85,B 0,C 180,E1 -11100.882,E2 -11100.882} C_VEL
LIN {X 0,Y 397.129,Z 364.64,A -85,B 0,C 180,E1 -11104.493,E2 -11104.493} C_VEL
LIN {X 0,Y 397.093,Z 364.645,A -85,B 0,C 180,E1 -11108.276,E2 -11108.276} C_VEL
LIN {X 0,Y 397.055,Z 364.65,A -85,B 0,C 180,E1 -11111.976,E2 -11111.976} C_VEL
LIN {X 0,Y 397.09,Z 364.641,A -85,B 0,C 180,E1 -11115.069,E2 -11115.069} C_VEL
LIN {X 0,Y 397.057,Z 364.65,A -85,B 0,C 180,E1 -11118.023,E2 -11118.023} C_VEL
LIN {X 0,Y 397.093,Z 364.644,A -85,B 0,C 180,E1 -11121.723,E2 -11121.723} C_VEL
LIN {X 0,Y 397.12,Z 364.639,A -85,B 0,C 180,E1 -11125.506,E2 -11125.506} C_VEL
LIN {X 0,Y 397.081,Z 364.649,A -85,B 0,C 180,E1 -11129.117,E2 -11129.117} C_VEL
LIN {X 0,Y 397.066,Z 364.625,A -85,B 0,C 180,E1 -11132.251,E2 -11132.251} C_VEL
LIN {X 0,Y 397.105,Z 364.613,A -85,B 0,C 180,E1 -11134.864,E2 -11134.864} C_VEL
LIN {X 0,Y 397.098,Z 364.643,A -85,B 0,C 180,E1 -11138.181,E2 -11138.181} C_VEL
LIN {X 0,Y 397.161,Z 364.633,A -85,B 0,C 180,E1 -11141.426,E2 -11141.426} C_VEL
LIN {X 0,Y 397.181,Z 364.63,A -85,B 0,C 180,E1 -11144.608,E2 -11144.608} C_VEL
LIN {X 0,Y 397.222,Z 364.619,A -85,B 0,C 180,E1 -11147.741,E2 -11147.741} C_VEL
LIN {X 0,Y 397.237,Z 364.623,A -85,B 0,C 180,E1 -11150.837,E2 -11150.837} C_VEL
LIN {X 0,Y 397.324,Z 364.607,A -85,B 0,C 180,E1 -11153.907,E2 -11153.907} C_VEL
LIN {X 0,Y 397.442,Z 364.602,A -85,B 0,C 180,E1 -11157.973,E2 -11157.973} C_VEL
LIN {X 0,Y 397.323,Z 364.609,A -85,B 0,C 180,E1 -11161.013,E2 -11161.013} C_VEL
LIN {X 0,Y 397.341,Z 364.607,A -85,B 0,C 180,E1 -11163.041,E2 -11163.041} C_VEL
LIN {X 0,Y 397.331,Z 364.612,A -85,B 0,C 180,E1 -11166.092,E2 -11166.092} C_VEL
LIN {X 0,Y 397.237,Z 364.622,A -85,B 0,C 180,E1 -11169.162,E2 -11169.162} C_VEL
LIN {X 0,Y 397.221,Z 364.621,A -85,B 0,C 180,E1 -11172.258,E2 -11172.258} C_VEL
LIN {X 0,Y 397.126,Z 364.64,A -85,B 0,C 180,E1 -11175.394,E2 -11175.394} C_VEL
LIN {X 0,Y 397.152,Z 364.63,A -85,B 0,C 180,E1 -11178.574,E2 -11178.574} C_VEL
LIN {X 0,Y 397.109,Z 364.638,A -85,B 0,C 180,E1 -11181.817,E2 -11181.817} C_VEL
LIN {X 0,Y 397.107,Z 364.642,A -85,B 0,C 180,E1 -11185.135,E2 -11185.135} C_VEL
LIN {X 0,Y 397.071,Z 364.646,A -85,B 0,C 180,E1 -11188.547,E2 -11188.547} C_VEL
LIN {X 0,Y 397.082,Z 364.648,A -85,B 0,C 180,E1 -11191.836,E2 -11191.836} C_VEL
LIN {X 0,Y 397.124,Z 364.64,A -85,B 0,C 180,E1 -11194.493,E2 -11194.493} C_VEL
LIN {X 0,Y 397.089,Z 364.64,A -85,B 0,C 180,E1 -11198.276,E2 -11198.276} C_VEL
LIN {X 0,Y 397.051,Z 364.651,A -85,B 0,C 180,E1 -11201.976,E2 -11201.976} C_VEL
LIN {X 0,Y 397.084,Z 364.647,A -85,B 0,C 180,E1 -11205.069,E2 -11205.069} C_VEL
LIN {X 0,Y 397.053,Z 364.655,A -85,B 0,C 180,E1 -11208.023,E2 -11208.023} C_VEL
LIN {X 0,Y 397.089,Z 364.647,A -85,B 0,C 180,E1 -11211.723,E2 -11211.723} C_VEL
LIN {X 0,Y 397.123,Z 364.645,A -85,B 0,C 180,E1 -11215.506,E2 -11215.506} C_VEL
LIN {X 0,Y 397.114,Z 364.718,A -85,B 0,C 180,E1 -11216.241,E2 -11216.241} C_VEL
LIN {X 0,Y 401.031,Z 380.599,A -85,B 0,C 180,E1 -11219.455,E2 -11219.455} C_VEL
LIN {X 0,Y 403.496,Z 392.093,A -85,B 0,C 180,E1 -11221.664,E2 -11221.664} C_VEL
LIN {X 0,Y 403.455,Z 394.462,A -85,B 0,C 180,E1 -11222.035,E2 -11222.035} C_VEL
LIN {X 0,Y 410.131,Z 430.09,A -85,B 0,C 180,E1 -11223.143,E2 -11223.143} C_VEL
LIN {X 0,Y 407.832,Z 558.588,A -85,B 0,C 180,E1 -11225.434,E2 -11225.434} C_VEL
LIN {X 0,Y 407.128,Z 573.761,A -85,B 0,C 180,E1 -11225.861,E2 -11225.861} C_VEL
LIN {X 0,Y 406.218,Z 587.708,A -85,B 0,C 180,E1 -11226.43,E2 -11226.43} C_VEL
LIN {X 0,Y 405.189,Z 601.817,A -85,B 0,C 180,E1 -11227.2,E2 -11227.2} C_VEL
LIN {X 0,Y 403.9,Z 615.757,A -85,B 0,C 180,E1 -11228.165,E2 -11228.165} C_VEL
LIN {X 0,Y 402.61,Z 628.915,A -85,B 0,C 180,E1 -11229.299,E2 -11229.299} C_VEL
LIN {X 0,Y 401.22,Z 641.035,A -85,B 0,C 180,E1 -11230.56,E2 -11230.56} C_VEL
LIN {X 0,Y 400.166,Z 651.337,A -85,B 0,C 180,E1 -11231.836,E2 -11231.836} C_VEL
LIN {X 0,Y 399.025,Z 661.767,A -85,B 0,C 180,E1 -11233.369,E2 -11233.369} C_VEL
LIN {X 0,Y 397.974,Z 671.977,A -85,B 0,C 180,E1 -11235.163,E2 -11235.163} C_VEL
LIN {X 0,Y 397.137,Z 680.112,A -85,B 0,C 180,E1 -11236.885,E2 -11236.885} C_VEL
LIN {X 0,Y 396.571,Z 687.459,A -85,B 0,C 180,E1 -11238.759,E2 -11238.759} C_VEL
LIN {X 0,Y 396.102,Z 693.956,A -85,B 0,C 180,E1 -11240.811,E2 -11240.811} C_VEL
LIN {X 0,Y 395.905,Z 699.004,A -85,B 0,C 180,E1 -11242.862,E2 -11242.862} C_VEL
LIN {X 0,Y 395.77,Z 702.731,A -85,B 0,C 180,E1 -11244.906,E2 -11244.906} C_VEL
LIN {X 0,Y 395.72,Z 705.227,A -85,B 0,C 180,E1 -11246.946,E2 -11246.946} C_VEL
LIN {X 0,Y 395.791,Z 706.515,A -85,B 0,C 180,E1 -11248.982,E2 -11248.982} C_VEL
LIN {X 0,Y 395.791,Z 706.623,A -85,B 0,C 180,E1 -11251.017,E2 -11251.017} C_VEL
LIN {X 0,Y 395.716,Z 705.593,A -85,B 0,C 180,E1 -11253.054,E2 -11253.054} C_VEL
LIN {X 0,Y 395.756,Z 703.419,A -85,B 0,C 180,E1 -11255.094,E2 -11255.094} C_VEL
LIN {X 0,Y 395.899,Z 700.058,A -85,B 0,C 180,E1 -11257.138,E2 -11257.138} C_VEL
LIN {X 0,Y 396.153,Z 695.408,A -85,B 0,C 180,E1 -11259.187,E2 -11259.187} C_VEL
LIN {X 0,Y 396.676,Z 689.366,A -85,B 0,C 180,E1 -11261.238,E2 -11261.238} C_VEL
LIN {X 0,Y 397.308,Z 681.507,A -85,B 0,C 180,E1 -11263.371,E2 -11263.371} C_VEL
LIN {X 0,Y 398.462,Z 672.501,A -85,B 0,C 180,E1 -11265.341,E2 -11265.341} C_VEL
LIN {X 0,Y 399.693,Z 662.602,A -85,B 0,C 180,E1 -11267.129,E2 -11267.129} C_VEL
LIN {X 0,Y 401.169,Z 651.695,A -85,B 0,C 180,E1 -11268.763,E2 -11268.763} C_VEL
LIN {X 0,Y 402.709,Z 639.427,A -85,B 0,C 180,E1 -11270.295,E2 -11270.295} C_VEL
LIN {X 0,Y 404.419,Z 625.916,A -85,B 0,C 180,E1 -11271.671,E2 -11271.671} C_VEL
LIN {X 0,Y 406.047,Z 612.409,A -85,B 0,C 180,E1 -11272.785,E2 -11272.785} C_VEL
LIN {X 0,Y 407.504,Z 597.483,A -85,B 0,C 180,E1 -11273.768,E2 -11273.768} C_VEL
LIN {X 0,Y 408.694,Z 582.786,A -85,B 0,C 180,E1 -11274.51,E2 -11274.51} C_VEL
LIN {X 0,Y 409.701,Z 567.771,A -85,B 0,C 180,E1 -11275.055,E2 -11275.055} C_VEL
LIN {X 0,Y 410.378,Z 552.166,A -85,B 0,C 180,E1 -11275.418,E2 -11275.418} C_VEL
LIN {X 0,Y 412.925,Z 431.328,A -85,B 0,C 180,E1 -11277.594,E2 -11277.594} C_VEL
LIN {X 0,Y 408.956,Z 410.184,A -85,B 0,C 180,E1 -11278.345,E2 -11278.345} C_VEL
LIN {X 0,Y 405.511,Z 396.138,A -85,B 0,C 180,E1 -11278.925,E2 -11278.925} C_VEL
LIN {X 0,Y 404.598,Z 393.769,A -85,B 0,C 180,E1 -11279.054,E2 -11279.054} C_VEL
LIN {X 0,Y 402.075,Z 382.578,A -85,B 0,C 180,E1 -11281.396,E2 -11281.396} C_VEL
LIN {X 0,Y 398.493,Z 369.333,A -85,B 0,C 180,E1 -11284.358,E2 -11284.358} C_VEL
LIN {X 0,Y 397.12,Z 364.644,A -85,B 0,C 180,E1 -11285.504,E2 -11285.504} C_VEL
LIN {X 0,Y 397.09,Z 364.638,A -85,B 0,C 180,E1 -11288.855,E2 -11288.855} C_VEL
LIN {X 0,Y 397.055,Z 364.643,A -85,B 0,C 180,E1 -11292.269,E2 -11292.269} C_VEL
LIN {X 0,Y 397.084,Z 364.648,A -85,B 0,C 180,E1 -11295.069,E2 -11295.069} C_VEL
LIN {X 0,Y 397.051,Z 364.651,A -85,B 0,C 180,E1 -11298.024,E2 -11298.024} C_VEL
LIN {X 0,Y 397.089,Z 364.646,A -85,B 0,C 180,E1 -11301.724,E2 -11301.724} C_VEL
LIN {X 0,Y 397.124,Z 364.637,A -85,B 0,C 180,E1 -11305.507,E2 -11305.507} C_VEL
LIN {X 0,Y 397.077,Z 364.625,A -85,B 0,C 180,E1 -11309.118,E2 -11309.118} C_VEL
LIN {X 0,Y 397.101,Z 364.644,A -85,B 0,C 180,E1 -11312.603,E2 -11312.603} C_VEL
LIN {X 0,Y 397.123,Z 364.643,A -85,B 0,C 180,E1 -11315.982,E2 -11315.982} C_VEL
LIN {X 0,Y 397.139,Z 364.638,A -85,B 0,C 180,E1 -11319.705,E2 -11319.705} C_VEL
LIN {X 0,Y 397.183,Z 364.633,A -85,B 0,C 180,E1 -11322.845,E2 -11322.845} C_VEL
LIN {X 0,Y 397.23,Z 364.626,A -85,B 0,C 180,E1 -11326.703,E2 -11326.703} C_VEL
LIN {X 0,Y 397.217,Z 364.629,A -85,B 0,C 180,E1 -11329.809,E2 -11329.809} C_VEL
LIN {X 0,Y 397.296,Z 364.621,A -85,B 0,C 180,E1 -11332.887,E2 -11332.887} C_VEL
LIN {X 0,Y 397.242,Z 364.621,A -85,B 0,C 180,E1 -11334.925,E2 -11334.925} C_VEL
LIN {X 0,Y 397.448,Z 364.602,A -85,B 0,C 180,E1 -11337.974,E2 -11337.974} C_VEL
LIN {X 0,Y 397.369,Z 364.611,A -85,B 0,C 180,E1 -11341.014,E2 -11341.014} C_VEL
LIN {X 0,Y 397.337,Z 364.608,A -85,B 0,C 180,E1 -11343.042,E2 -11343.042} C_VEL
LIN {X 0,Y 397.301,Z 364.615,A -85,B 0,C 180,E1 -11346.554,E2 -11346.554} C_VEL
LIN {X 0,Y 397.237,Z 364.627,A -85,B 0,C 180,E1 -11349.163,E2 -11349.163} C_VEL
LIN {X 0,Y 397.221,Z 364.628,A -85,B 0,C 180,E1 -11352.259,E2 -11352.259} C_VEL
LIN {X 0,Y 397.181,Z 364.631,A -85,B 0,C 180,E1 -11355.392,E2 -11355.392} C_VEL
LIN {X 0,Y 397.163,Z 364.62,A -85,B 0,C 180,E1 -11358.574,E2 -11358.574} C_VEL
LIN {X 0,Y 397.098,Z 364.64,A -85,B 0,C 180,E1 -11361.819,E2 -11361.819} C_VEL
LIN {X 0,Y 397.1,Z 364.627,A -85,B 0,C 180,E1 -11365.136,E2 -11365.136} C_VEL
LIN {X 0,Y 397.102,Z 364.648,A -85,B 0,C 180,E1 -11368.546,E2 -11368.546} C_VEL
LIN {X 0,Y 397.081,Z 364.638,A -85,B 0,C 180,E1 -11372.072,E2 -11372.072} C_VEL
LIN {X 0,Y 397.125,Z 364.635,A -85,B 0,C 180,E1 -11374.494,E2 -11374.494} C_VEL
LIN {X 0,Y 397.093,Z 364.643,A -85,B 0,C 180,E1 -11378.277,E2 -11378.277} C_VEL
LIN {X 0,Y 397.056,Z 364.647,A -85,B 0,C 180,E1 -11381.977,E2 -11381.977} C_VEL
LIN {X 0,Y 397.089,Z 364.641,A -85,B 0,C 180,E1 -11385.069,E2 -11385.069} C_VEL
LIN {X 0,Y 397.084,Z 364.716,A -85,B 0,C 180,E1 -11388.381,E2 -11388.381} C_VEL
LIN {X 0,Y 399.51,Z 373.515,A -85,B 0,C 180,E1 -11390.537,E2 -11390.537} C_VEL
LIN {X 0,Y 408.679,Z 392.021,A -85,B 0,C 180,E1 -11391.736,E2 -11391.736} C_VEL
LIN {X 0,Y 413.387,Z 402.981,A -85,B 0,C 180,E1 -11392.352,E2 -11392.352} C_VEL
LIN {X 0,Y 411.755,Z 477.562,A -85,B 0,C 180,E1 -11393.697,E2 -11393.697} C_VEL
LIN {X 0,Y 410.387,Z 536.332,A -85,B 0,C 180,E1 -11394.767,E2 -11394.767} C_VEL
LIN {X 0,Y 409.705,Z 551.826,A -85,B 0,C 180,E1 -11395.224,E2 -11395.224} C_VEL
LIN {X 0,Y 408.762,Z 566.856,A -85,B 0,C 180,E1 -11395.877,E2 -11395.877} C_VEL
LIN {X 0,Y 407.53,Z 580.474,A -85,B 0,C 180,E1 -11396.654,E2 -11396.654} C_VEL
LIN {X 0,Y 406.276,Z 594.279,A -85,B 0,C 180,E1 -11397.665,E2 -11397.665} C_VEL
LIN {X 0,Y 404.887,Z 606.573,A -85,B 0,C 180,E1 -11398.764,E2 -11398.764} C_VEL
LIN {X 0,Y 403.295,Z 618.783,A -85,B 0,C 180,E1 -11400.077,E2 -11400.077} C_VEL
LIN {X 0,Y 401.829,Z 630.121,A -85,B 0,C 180,E1 -11401.552,E2 -11401.552} C_VEL
LIN {X 0,Y 400.518,Z 640.107,A -85,B 0,C 180,E1 -11403.101,E2 -11403.101} C_VEL
LIN {X 0,Y 399.259,Z 649.001,A -85,B 0,C 180,E1 -11404.731,E2 -11404.731} C_VEL
LIN {X 0,Y 398.105,Z 657.599,A -85,B 0,C 180,E1 -11406.635,E2 -11406.635} C_VEL
LIN {X 0,Y 397.392,Z 663.436,A -85,B 0,C 180,E1 -11408.199,E2 -11408.199} C_VEL
LIN {X 0,Y 396.642,Z 669.987,A -85,B 0,C 180,E1 -11410.327,E2 -11410.327} C_VEL
LIN {X 0,Y 396.173,Z 675.007,A -85,B 0,C 180,E1 -11412.448,E2 -11412.448} C_VEL
LIN {X 0,Y 395.896,Z 678.648,A -85,B 0,C 180,E1 -11414.557,E2 -11414.557} C_VEL
LIN {X 0,Y 395.75,Z 681.025,A -85,B 0,C 180,E1 -11416.652,E2 -11416.652} C_VEL
LIN {X 0,Y 395.699,Z 682.208,A -85,B 0,C 180,E1 -11418.734,E2 -11418.734} C_VEL
LIN {X 0,Y 395.64,Z 682.199,A -85,B 0,C 180,E1 -11420.801,E2 -11420.801} C_VEL
LIN {X 0,Y 395.767,Z 681.014,A -85,B 0,C 180,E1 -11422.859,E2 -11422.859} C_VEL
LIN {X 0,Y 395.89,Z 678.682,A -85,B 0,C 180,E1 -11424.908,E2 -11424.908} C_VEL
LIN {X 0,Y 395.896,Z 677.918,A -85,B 0,C 180,E1 -11425.393,E2 -11425.393} C_VEL
LIN {X 0,Y 395.277,Z 676.611,A -85,B 0,C 180,E1 -11426.221,E2 -11426.221} C_VEL
LIN {X 0,Y 392.54,Z 674.098,A -85,B 0,C 180,E1 -11427.56,E2 -11427.56} C_VEL
LIN {X 0,Y 390.272,Z 671.753,A -85,B 0,C 180,E1 -11428.626,E2 -11428.626} C_VEL
LIN {X 0,Y 389.385,Z 669.691,A -85,B 0,C 180,E1 -11429.436,E2 -11429.436} C_VEL
LIN {X 0,Y 389.359,Z 668.947,A -85,B 0,C 180,E1 -11429.707,E2 -11429.707} C_VEL
LIN {X 0,Y 389.983,Z 663.126,A -85,B 0,C 180,E1 -11431.549,E2 -11431.549} C_VEL
LIN {X 0,Y 390.867,Z 655.097,A -85,B 0,C 180,E1 -11433.608,E2 -11433.608} C_VEL
LIN {X 0,Y 391.837,Z 646.557,A -85,B 0,C 180,E1 -11435.403,E2 -11435.403} C_VEL
LIN {X 0,Y 393.054,Z 636.31,A -85,B 0,C 180,E1 -11437.19,E2 -11437.19} C_VEL
LIN {X 0,Y 394.35,Z 625.817,A -85,B 0,C 180,E1 -11438.713,E2 -11438.713} C_VEL
LIN {X 0,Y 395.768,Z 613.267,A -85,B 0,C 180,E1 -11440.229,E2 -11440.229} C_VEL
LIN {X 0,Y 397.058,Z 600.656,A -85,B 0,C 180,E1 -11441.486,E2 -11441.486} C_VEL
LIN {X 0,Y 398.421,Z 586.762,A -85,B 0,C 180,E1 -11442.609,E2 -11442.609} C_VEL
LIN {X 0,Y 399.472,Z 573.332,A -85,B 0,C 180,E1 -11443.48,E2 -11443.48} C_VEL
LIN {X 0,Y 400.474,Z 558.425,A -85,B 0,C 180,E1 -11444.223,E2 -11444.223} C_VEL
LIN {X 0,Y 401.14,Z 543.929,A -85,B 0,C 180,E1 -11444.749,E2 -11444.749} C_VEL
LIN {X 0,Y 401.671,Z 527.808,A -85,B 0,C 180,E1 -11445.118,E2 -11445.118} C_VEL
LIN {X 0,Y 404.029,Z 403.647,A -85,B 0,C 180,E1 -11447.349,E2 -11447.349} C_VEL
LIN {X 0,Y 402.745,Z 399.173,A -85,B 0,C 180,E1 -11447.52,E2 -11447.52} C_VEL
LIN {X 0,Y 393.297,Z 376.258,A -85,B 0,C 180,E1 -11448.615,E2 -11448.615} C_VEL
LIN {X 0,Y 391.892,Z 372.961,A -85,B 0,C 180,E1 -11448.786,E2 -11448.786} C_VEL
LIN {X 0,Y 390.099,Z 365.51,A -85,B 0,C 180,E1 -11450.518,E2 -11450.518} C_VEL
LIN {X 0,Y 390.067,Z 365.522,A -85,B 0,C 180,E1 -11453.352,E2 -11453.352} C_VEL
LIN {X 0,Y 390.047,Z 365.523,A -85,B 0,C 180,E1 -11456.773,E2 -11456.773} C_VEL
LIN {X 0,Y 390.041,Z 365.522,A -85,B 0,C 180,E1 -11460.3,E2 -11460.3} C_VEL
LIN {X 0,Y 390.073,Z 365.521,A -85,B 0,C 180,E1 -11464.024,E2 -11464.024} C_VEL
LIN {X 0,Y 390.041,Z 365.523,A -85,B 0,C 180,E1 -11467.549,E2 -11467.549} C_VEL
LIN {X 0,Y 390.02,Z 365.515,A -85,B 0,C 180,E1 -11470.814,E2 -11470.814} C_VEL
LIN {X 0,Y 390.055,Z 365.52,A -85,B 0,C 180,E1 -11473.885,E2 -11473.885} C_VEL
LIN {X 0,Y 390.056,Z 365.51,A -85,B 0,C 180,E1 -11476.789,E2 -11476.789} C_VEL
LIN {X 0,Y 390.013,Z 365.53,A -85,B 0,C 180,E1 -11479.554,E2 -11479.554} C_VEL
LIN {X 0,Y 390.041,Z 365.522,A -85,B 0,C 180,E1 -11482.45,E2 -11482.45} C_VEL
LIN {X 0,Y 390.064,Z 365.517,A -85,B 0,C 180,E1 -11486.044,E2 -11486.044} C_VEL
LIN {X 0,Y 390.047,Z 365.52,A -85,B 0,C 180,E1 -11489.87,E2 -11489.87} C_VEL
LIN {X 0,Y 390.034,Z 365.49,A -85,B 0,C 180,E1 -11493.225,E2 -11493.225} C_VEL
LIN {X 0,Y 390.068,Z 365.509,A -85,B 0,C 180,E1 -11496.764,E2 -11496.764} C_VEL
LIN {X 0,Y 390.11,Z 365.514,A -85,B 0,C 180,E1 -11499.983,E2 -11499.983} C_VEL
LIN {X 0,Y 390.141,Z 365.501,A -85,B 0,C 180,E1 -11503.248,E2 -11503.248} C_VEL
LIN {X 0,Y 390.198,Z 365.5,A -85,B 0,C 180,E1 -11506.561,E2 -11506.561} C_VEL
LIN {X 0,Y 390.168,Z 365.5,A -85,B 0,C 180,E1 -11509.622,E2 -11509.622} C_VEL
LIN {X 0,Y 390.249,Z 365.494,A -85,B 0,C 180,E1 -11512.757,E2 -11512.757} C_VEL
LIN {X 0,Y 390.203,Z 365.491,A -85,B 0,C 180,E1 -11514.833,E2 -11514.833} C_VEL
LIN {X 0,Y 390.41,Z 365.478,A -85,B 0,C 180,E1 -11517.936,E2 -11517.936} C_VEL
LIN {X 0,Y 390.294,Z 365.485,A -85,B 0,C 180,E1 -11521.031,E2 -11521.031} C_VEL
LIN {X 0,Y 390.277,Z 365.487,A -85,B 0,C 180,E1 -11523.096,E2 -11523.096} C_VEL
LIN {X 0,Y 390.285,Z 365.489,A -85,B 0,C 180,E1 -11526.202,E2 -11526.202} C_VEL
LIN {X 0,Y 390.194,Z 365.501,A -85,B 0,C 180,E1 -11529.329,E2 -11529.329} C_VEL
LIN {X 0,Y 390.172,Z 365.498,A -85,B 0,C 180,E1 -11532.483,E2 -11532.483} C_VEL
LIN {X 0,Y 390.069,Z 365.521,A -85,B 0,C 180,E1 -11535.679,E2 -11535.679} C_VEL
LIN {X 0,Y 390.099,Z 365.509,A -85,B 0,C 180,E1 -11538.922,E2 -11538.922} C_VEL
LIN {X 0,Y 390.045,Z 365.516,A -85,B 0,C 180,E1 -11542.233,E2 -11542.233} C_VEL
LIN {X 0,Y 390.05,Z 365.52,A -85,B 0,C 180,E1 -11545.722,E2 -11545.722} C_VEL
LIN {X 0,Y 390.029,Z 365.525,A -85,B 0,C 180,E1 -11549.112,E2 -11549.112} C_VEL
LIN {X 0,Y 390.043,Z 365.52,A -85,B 0,C 180,E1 -11552.721,E2 -11552.721} C_VEL
LIN {X 0,Y 390.054,Z 365.522,A -85,B 0,C 180,E1 -11555.824,E2 -11555.824} C_VEL
LIN {X 0,Y 390.035,Z 365.517,A -85,B 0,C 180,E1 -11559.212,E2 -11559.212} C_VEL
LIN {X 0,Y 390.029,Z 365.523,A -85,B 0,C 180,E1 -11562.372,E2 -11562.372} C_VEL
LIN {X 0,Y 390.041,Z 365.526,A -85,B 0,C 180,E1 -11565.354,E2 -11565.354} C_VEL
LIN {X 0,Y 390.016,Z 365.53,A -85,B 0,C 180,E1 -11568.184,E2 -11568.184} C_VEL
LIN {X 0,Y 390.056,Z 365.526,A -85,B 0,C 180,E1 -11570.903,E2 -11570.903} C_VEL
LIN {X 0,Y 390.083,Z 365.52,A -85,B 0,C 180,E1 -11574.793,E2 -11574.793} C_VEL
LIN {X 0,Y 390.096,Z 365.625,A -85,B 0,C 180,E1 -11575.844,E2 -11575.844} C_VEL
LIN {X 0,Y 394.029,Z 381.736,A -85,B 0,C 180,E1 -11579.174,E2 -11579.174} C_VEL
LIN {X 0,Y 396.657,Z 393.902,A -85,B 0,C 180,E1 -11581.558,E2 -11581.558} C_VEL
LIN {X 0,Y 403.651,Z 431.127,A -85,B 0,C 180,E1 -11582.754,E2 -11582.754} C_VEL
LIN {X 0,Y 401.218,Z 559.088,A -85,B 0,C 180,E1 -11585.071,E2 -11585.071} C_VEL
LIN {X 0,Y 400.45,Z 575.004,A -85,B 0,C 180,E1 -11585.539,E2 -11585.539} C_VEL
LIN {X 0,Y 399.505,Z 588.861,A -85,B 0,C 180,E1 -11586.133,E2 -11586.133} C_VEL
LIN {X 0,Y 398.386,Z 603.042,A -85,B 0,C 180,E1 -11586.938,E2 -11586.938} C_VEL
LIN {X 0,Y 397.085,Z 616.544,A -85,B 0,C 180,E1 -11587.907,E2 -11587.907} C_VEL
LIN {X 0,Y 395.75,Z 629.522,A -85,B 0,C 180,E1 -11589.06,E2 -11589.06} C_VEL
LIN {X 0,Y 394.316,Z 641.506,A -85,B 0,C 180,E1 -11590.341,E2 -11590.341} C_VEL
LIN {X 0,Y 393.134,Z 652.619,A -85,B 0,C 180,E1 -11591.769,E2 -11591.769} C_VEL
LIN {X 0,Y 391.923,Z 662.856,A -85,B 0,C 180,E1 -11593.327,E2 -11593.327} C_VEL
LIN {X 0,Y 390.896,Z 672.843,A -85,B 0,C 180,E1 -11595.155,E2 -11595.155} C_VEL
LIN {X 0,Y 390.026,Z 681.376,A -85,B 0,C 180,E1 -11597.038,E2 -11597.038} C_VEL
LIN {X 0,Y 389.377,Z 688.902,A -85,B 0,C 180,E1 -11599.075,E2 -11599.075} C_VEL
LIN {X 0,Y 388.975,Z 695.055,A -85,B 0,C 180,E1 -11601.166,E2 -11601.166} C_VEL
LIN {X 0,Y 388.762,Z 699.774,A -85,B 0,C 180,E1 -11603.252,E2 -11603.252} C_VEL
LIN {X 0,Y 388.674,Z 702.451,A -85,B 0,C 180,E1 -11604.813,E2 -11604.813} C_VEL
LIN {X 0,Y 388.627,Z 704.975,A -85,B 0,C 180,E1 -11606.89,E2 -11606.89} C_VEL
LIN {X 0,Y 388.722,Z 706.277,A -85,B 0,C 180,E1 -11608.964,E2 -11608.964} C_VEL
LIN {X 0,Y 388.721,Z 706.411,A -85,B 0,C 180,E1 -11611.036,E2 -11611.036} C_VEL
LIN {X 0,Y 388.622,Z 705.406,A -85,B 0,C 180,E1 -11613.11,E2 -11613.11} C_VEL
LIN {X 0,Y 388.662,Z 703.259,A -85,B 0,C 180,E1 -11615.187,E2 -11615.187} C_VEL
LIN {X 0,Y 388.819,Z 699.926,A -85,B 0,C 180,E1 -11617.269,E2 -11617.269} C_VEL
LIN {X 0,Y 389.076,Z 695.292,A -85,B 0,C 180,E1 -11619.356,E2 -11619.356} C_VEL
LIN {X 0,Y 389.646,Z 689.284,A -85,B 0,C 180,E1 -11621.444,E2 -11621.444} C_VEL
LIN {X 0,Y 390.313,Z 681.762,A -85,B 0,C 180,E1 -11623.537,E2 -11623.537} C_VEL
LIN {X 0,Y 391.564,Z 672.504,A -85,B 0,C 180,E1 -11625.618,E2 -11625.618} C_VEL
LIN {X 0,Y 392.874,Z 662.654,A -85,B 0,C 180,E1 -11627.436,E2 -11627.436} C_VEL
LIN {X 0,Y 394.34,Z 652.367,A -85,B 0,C 180,E1 -11629.015,E2 -11629.015} C_VEL
LIN {X 0,Y 395.878,Z 640.675,A -85,B 0,C 180,E1 -11630.525,E2 -11630.525} C_VEL
LIN {X 0,Y 397.485,Z 628.797,A -85,B 0,C 180,E1 -11631.796,E2 -11631.796} C_VEL
LIN {X 0,Y 399.131,Z 615.97,A -85,B 0,C 180,E1 -11632.929,E2 -11632.929} C_VEL
LIN {X 0,Y 400.628,Z 602.49,A -85,B 0,C 180,E1 -11633.897,E2 -11633.897} C_VEL
LIN {X 0,Y 401.912,Z 588.102,A -85,B 0,C 180,E1 -11634.715,E2 -11634.715} C_VEL
LIN {X 0,Y 403.046,Z 573.583,A -85,B 0,C 180,E1 -11635.325,E2 -11635.325} C_VEL
LIN {X 0,Y 403.896,Z 558.831,A -85,B 0,C 180,E1 -11635.752,E2 -11635.752} C_VEL
LIN {X 0,Y 406.782,Z 432.249,A -85,B 0,C 180,E1 -11638.082,E2 -11638.082} C_VEL
LIN {X 0,Y 402.731,Z 410.829,A -85,B 0,C 180,E1 -11638.866,E2 -11638.866} C_VEL
LIN {X 0,Y 399.897,Z 399.278,A -85,B 0,C 180,E1 -11639.358,E2 -11639.358} C_VEL
LIN {X 0,Y 397.43,Z 393.432,A -85,B 0,C 180,E1 -11639.719,E2 -11639.719} C_VEL
LIN {X 0,Y 394.857,Z 382.777,A -85,B 0,C 180,E1 -11642.025,E2 -11642.025} C_VEL
LIN {X 0,Y 391.406,Z 370.217,A -85,B 0,C 180,E1 -11644.925,E2 -11644.925} C_VEL
LIN {X 0,Y 390.06,Z 365.517,A -85,B 0,C 180,E1 -11646.11,E2 -11646.11} C_VEL
LIN {X 0,Y 390.035,Z 365.517,A -85,B 0,C 180,E1 -11649.212,E2 -11649.212} C_VEL
LIN {X 0,Y 390.031,Z 365.518,A -85,B 0,C 180,E1 -11652.373,E2 -11652.373} C_VEL
LIN {X 0,Y 390.041,Z 365.524,A -85,B 0,C 180,E1 -11655.354,E2 -11655.354} C_VEL
LIN {X 0,Y 390.014,Z 365.528,A -85,B 0,C 180,E1 -11658.185,E2 -11658.185} C_VEL
LIN {X 0,Y 390.056,Z 365.523,A -85,B 0,C 180,E1 -11660.904,E2 -11660.904} C_VEL
LIN {X 0,Y 390.084,Z 365.508,A -85,B 0,C 180,E1 -11664.793,E2 -11664.793} C_VEL
LIN {X 0,Y 390.023,Z 365.507,A -85,B 0,C 180,E1 -11668.496,E2 -11668.496} C_VEL
LIN {X 0,Y 390.038,Z 365.524,A -85,B 0,C 180,E1 -11672.064,E2 -11672.064} C_VEL
LIN {X 0,Y 390.06,Z 365.521,A -85,B 0,C 180,E1 -11675.518,E2 -11675.518} C_VEL
LIN {X 0,Y 390.063,Z 365.522,A -85,B 0,C 180,E1 -11678.879,E2 -11678.879} C_VEL
LIN {X 0,Y 390.126,Z 365.515,A -85,B 0,C 180,E1 -11682.167,E2 -11682.167} C_VEL
LIN {X 0,Y 390.143,Z 365.509,A -85,B 0,C 180,E1 -11685.393,E2 -11685.393} C_VEL
LIN {X 0,Y 390.148,Z 365.509,A -85,B 0,C 180,E1 -11688.572,E2 -11688.572} C_VEL
LIN {X 0,Y 390.258,Z 365.491,A -85,B 0,C 180,E1 -11692.086,E2 -11692.086} C_VEL
LIN {X 0,Y 390.212,Z 365.497,A -85,B 0,C 180,E1 -11694.834,E2 -11694.834} C_VEL
LIN {X 0,Y 390.417,Z 365.478,A -85,B 0,C 180,E1 -11697.937,E2 -11697.937} C_VEL
LIN {X 0,Y 390.336,Z 365.487,A -85,B 0,C 180,E1 -11701.032,E2 -11701.032} C_VEL
LIN {X 0,Y 390.273,Z 365.487,A -85,B 0,C 180,E1 -11703.097,E2 -11703.097} C_VEL
LIN {X 0,Y 390.261,Z 365.494,A -85,B 0,C 180,E1 -11706.545,E2 -11706.545} C_VEL
LIN {X 0,Y 390.195,Z 365.504,A -85,B 0,C 180,E1 -11709.33,E2 -11709.33} C_VEL
LIN {X 0,Y 390.173,Z 365.509,A -85,B 0,C 180,E1 -11712.484,E2 -11712.484} C_VEL
LIN {X 0,Y 390.142,Z 365.509,A -85,B 0,C 180,E1 -11715.677,E2 -11715.677} C_VEL
LIN {X 0,Y 390.107,Z 365.495,A -85,B 0,C 180,E1 -11718.923,E2 -11718.923} C_VEL
LIN {X 0,Y 390.039,Z 365.523,A -85,B 0,C 180,E1 -11722.235,E2 -11722.235} C_VEL
LIN {X 0,Y 390.052,Z 365.502,A -85,B 0,C 180,E1 -11725.722,E2 -11725.722} C_VEL
LIN {X 0,Y 390.046,Z 365.521,A -85,B 0,C 180,E1 -11729.111,E2 -11729.111} C_VEL
LIN {X 0,Y 390.046,Z 365.523,A -85,B 0,C 180,E1 -11732.722,E2 -11732.722} C_VEL
LIN {X 0,Y 390.047,Z 365.51,A -85,B 0,C 180,E1 -11735.823,E2 -11735.823} C_VEL
LIN {X 0,Y 390.038,Z 365.514,A -85,B 0,C 180,E1 -11739.212,E2 -11739.212} C_VEL
LIN {X 0,Y 390.035,Z 365.519,A -85,B 0,C 180,E1 -11742.373,E2 -11742.373} C_VEL
LIN {X 0,Y 390.047,Z 365.518,A -85,B 0,C 180,E1 -11745.355,E2 -11745.355} C_VEL
LIN {X 0,Y 390.045,Z 365.612,A -85,B 0,C 180,E1 -11747.808,E2 -11747.808} C_VEL
LIN {X 0,Y 392.332,Z 373.763,A -85,B 0,C 180,E1 -11749.864,E2 -11749.864} C_VEL
LIN {X 0,Y 401.675,Z 392.289,A -85,B 0,C 180,E1 -11751.127,E2 -11751.127} C_VEL
LIN {X 0,Y 407.238,Z 404.625,A -85,B 0,C 180,E1 -11751.868,E2 -11751.868} C_VEL
LIN {X 0,Y 405.756,Z 471.515,A -85,B 0,C 180,E1 -11753.097,E2 -11753.097} C_VEL
LIN {X 0,Y 404.146,Z 536.52,A -85,B 0,C 180,E1 -11754.293,E2 -11754.293} C_VEL
LIN {X 0,Y 403.438,Z 552.022,A -85,B 0,C 180,E1 -11754.757,E2 -11754.757} C_VEL
LIN {X 0,Y 402.51,Z 566.274,A -85,B 0,C 180,E1 -11755.38,E2 -11755.38} C_VEL
LIN {X 0,Y 401.147,Z 580.664,A -85,B 0,C 180,E1 -11756.203,E2 -11756.203} C_VEL
LIN {X 0,Y 399.871,Z 594.362,A -85,B 0,C 180,E1 -11757.221,E2 -11757.221} C_VEL
LIN {X 0,Y 398.395,Z 606.768,A -85,B 0,C 180,E1 -11758.344,E2 -11758.344} C_VEL
LIN {X 0,Y 396.722,Z 618.976,A -85,B 0,C 180,E1 -11759.676,E2 -11759.676} C_VEL
LIN {X 0,Y 395.048,Z 631.13,A -85,B 0,C 180,E1 -11761.293,E2 -11761.293} C_VEL
LIN {X 0,Y 393.636,Z 641.273,A -85,B 0,C 180,E1 -11762.918,E2 -11762.918} C_VEL
LIN {X 0,Y 392.145,Z 651.098,A -85,B 0,C 180,E1 -11764.808,E2 -11764.808} C_VEL
LIN {X 0,Y 391.037,Z 659.207,A -85,B 0,C 180,E1 -11766.709,E2 -11766.709} C_VEL
LIN {X 0,Y 390.033,Z 666.701,A -85,B 0,C 180,E1 -11768.876,E2 -11768.876} C_VEL
LIN {X 0,Y 389.405,Z 672.566,A -85,B 0,C 180,E1 -11771.043,E2 -11771.043} C_VEL
LIN {X 0,Y 389.053,Z 677.008,A -85,B 0,C 180,E1 -11773.221,E2 -11773.221} C_VEL
LIN {X 0,Y 388.713,Z 680.061,A -85,B 0,C 180,E1 -11775.338,E2 -11775.338} C_VEL
LIN {X 0,Y 388.689,Z 681.945,A -85,B 0,C 180,E1 -11777.528,E2 -11777.528} C_VEL
LIN {X 0,Y 388.573,Z 682.562,A -85,B 0,C 180,E1 -11779.58,E2 -11779.58} C_VEL
LIN {X 0,Y 388.58,Z 682.033,A -85,B 0,C 180,E1 -11781.681,E2 -11781.681} C_VEL
LIN {X 0,Y 388.784,Z 680.278,A -85,B 0,C 180,E1 -11783.847,E2 -11783.847} C_VEL
LIN {X 0,Y 388.844,Z 677.529,A -85,B 0,C 180,E1 -11785.854,E2 -11785.854} C_VEL
LIN {X 0,Y 389.096,Z 673.48,A -85,B 0,C 180,E1 -11787.93,E2 -11787.93} C_VEL
LIN {X 0,Y 389.359,Z 668.947,A -85,B 0,C 180,E1 -11789.707,E2 -11789.707} C_VEL
LIN {X 0,Y 388.9,Z 666.667,A -85,B 0,C 180,E1 -11790.507,E2 -11790.507} C_VEL
LIN {X 0,Y 386.491,Z 662.682,A -85,B 0,C 180,E1 -11791.801,E2 -11791.801} C_VEL
LIN {X 0,Y 384.185,Z 658.264,A -85,B 0,C 180,E1 -11793.076,E2 -11793.076} C_VEL
LIN {X 0,Y 383.894,Z 655.21,A -85,B 0,C 180,E1 -11793.835,E2 -11793.835} C_VEL
LIN {X 0,Y 385,Z 646.123,A -85,B 0,C 180,E1 -11795.762,E2 -11795.762} C_VEL
LIN {X 0,Y 386.283,Z 635.742,A -85,B 0,C 180,E1 -11797.58,E2 -11797.58} C_VEL
LIN {X 0,Y 387.637,Z 625.093,A -85,B 0,C 180,E1 -11799.128,E2 -11799.128} C_VEL
LIN {X 0,Y 388.984,Z 613.507,A -85,B 0,C 180,E1 -11800.541,E2 -11800.541} C_VEL
LIN {X 0,Y 390.351,Z 600.889,A -85,B 0,C 180,E1 -11801.818,E2 -11801.818} C_VEL
LIN {X 0,Y 391.757,Z 586.994,A -85,B 0,C 180,E1 -11802.959,E2 -11802.959} C_VEL
LIN {X 0,Y 392.849,Z 573.562,A -85,B 0,C 180,E1 -11803.844,E2 -11803.844} C_VEL
LIN {X 0,Y 393.874,Z 558.661,A -85,B 0,C 180,E1 -11804.598,E2 -11804.598} C_VEL
LIN {X 0,Y 394.573,Z 544.164,A -85,B 0,C 180,E1 -11805.133,E2 -11805.133} C_VEL
LIN {X 0,Y 395.112,Z 528.416,A -85,B 0,C 180,E1 -11805.501,E2 -11805.501} C_VEL
LIN {X 0,Y 397.58,Z 404.817,A -85,B 0,C 180,E1 -11807.754,E2 -11807.754} C_VEL
LIN {X 0,Y 394.782,Z 397.085,A -85,B 0,C 180,E1 -11808.097,E2 -11808.097} C_VEL
LIN {X 0,Y 384.679,Z 373.2,A -85,B 0,C 180,E1 -11809.304,E2 -11809.304} C_VEL
LIN {X 0,Y 383.032,Z 366.389,A -85,B 0,C 180,E1 -11810.932,E2 -11810.932} C_VEL
LIN {X 0,Y 383.014,Z 366.403,A -85,B 0,C 180,E1 -11813.809,E2 -11813.809} C_VEL
LIN {X 0,Y 382.986,Z 366.406,A -85,B 0,C 180,E1 -11817.308,E2 -11817.308} C_VEL
LIN {X 0,Y 382.987,Z 366.402,A -85,B 0,C 180,E1 -11820.918,E2 -11820.918} C_VEL
LIN {X 0,Y 383.022,Z 366.397,A -85,B 0,C 180,E1 -11824.668,E2 -11824.668} C_VEL
LIN {X 0,Y 382.996,Z 366.404,A -85,B 0,C 180,E1 -11827.902,E2 -11827.902} C_VEL
LIN {X 0,Y 382.964,Z 366.396,A -85,B 0,C 180,E1 -11831.35,E2 -11831.35} C_VEL
LIN {X 0,Y 382.997,Z 366.397,A -85,B 0,C 180,E1 -11834.303,E2 -11834.303} C_VEL
LIN {X 0,Y 383.014,Z 366.39,A -85,B 0,C 180,E1 -11837.24,E2 -11837.24} C_VEL
LIN {X 0,Y 382.988,Z 366.397,A -85,B 0,C 180,E1 -11840.419,E2 -11840.419} C_VEL
LIN {X 0,Y 383.017,Z 366.398,A -85,B 0,C 180,E1 -11844.043,E2 -11844.043} C_VEL
LIN {X 0,Y 382.989,Z 366.405,A -85,B 0,C 180,E1 -11847.578,E2 -11847.578} C_VEL
LIN {X 0,Y 382.98,Z 366.397,A -85,B 0,C 180,E1 -11850.298,E2 -11850.298} C_VEL
LIN {X 0,Y 383.005,Z 366.363,A -85,B 0,C 180,E1 -11854.045,E2 -11854.045} C_VEL
LIN {X 0,Y 382.992,Z 366.394,A -85,B 0,C 180,E1 -11857.334,E2 -11857.334} C_VEL
LIN {X 0,Y 383.063,Z 366.39,A -85,B 0,C 180,E1 -11860.716,E2 -11860.716} C_VEL
LIN {X 0,Y 383.084,Z 366.389,A -85,B 0,C 180,E1 -11864.026,E2 -11864.026} C_VEL
LIN {X 0,Y 383.139,Z 366.38,A -85,B 0,C 180,E1 -11867.283,E2 -11867.283} C_VEL
LIN {X 0,Y 383.145,Z 366.378,A -85,B 0,C 180,E1 -11870.497,E2 -11870.497} C_VEL
LIN {X 0,Y 383.237,Z 366.364,A -85,B 0,C 180,E1 -11873.682,E2 -11873.682} C_VEL
LIN {X 0,Y 383.376,Z 366.355,A -85,B 0,C 180,E1 -11877.898,E2 -11877.898} C_VEL
LIN {X 0,Y 383.265,Z 366.36,A -85,B 0,C 180,E1 -11881.05,E2 -11881.05} C_VEL
LIN {X 0,Y 383.382,Z 366.345,A -85,B 0,C 180,E1 -11882.101,E2 -11882.101} C_VEL
LIN {X 0,Y 383.242,Z 366.366,A -85,B 0,C 180,E1 -11886.317,E2 -11886.317} C_VEL
LIN {X 0,Y 383.145,Z 366.381,A -85,B 0,C 180,E1 -11889.502,E2 -11889.502} C_VEL
LIN {X 0,Y 383.127,Z 366.378,A -85,B 0,C 180,E1 -11893.536,E2 -11893.536} C_VEL
LIN {X 0,Y 383.059,Z 366.388,A -85,B 0,C 180,E1 -11897.436,E2 -11897.436} C_VEL
LIN {X 0,Y 383.032,Z 366.392,A -85,B 0,C 180,E1 -11900.647,E2 -11900.647} C_VEL
LIN {X 0,Y 383.014,Z 366.401,A -85,B 0,C 180,E1 -11903.808,E2 -11903.808} C_VEL
LIN {X 0,Y 382.985,Z 366.4,A -85,B 0,C 180,E1 -11907.307,E2 -11907.307} C_VEL
LIN {X 0,Y 382.982,Z 366.401,A -85,B 0,C 180,E1 -11910.918,E2 -11910.918} C_VEL
LIN {X 0,Y 383.018,Z 366.397,A -85,B 0,C 180,E1 -11914.668,E2 -11914.668} C_VEL
LIN {X 0,Y 382.991,Z 366.399,A -85,B 0,C 180,E1 -11917.902,E2 -11917.902} C_VEL
LIN {X 0,Y 382.959,Z 366.406,A -85,B 0,C 180,E1 -11921.35,E2 -11921.35} C_VEL
LIN {X 0,Y 382.992,Z 366.402,A -85,B 0,C 180,E1 -11924.302,E2 -11924.302} C_VEL
LIN {X 0,Y 383.01,Z 366.403,A -85,B 0,C 180,E1 -11927.24,E2 -11927.24} C_VEL
LIN {X 0,Y 382.984,Z 366.407,A -85,B 0,C 180,E1 -11930.419,E2 -11930.419} C_VEL
LIN {X 0,Y 383.022,Z 366.398,A -85,B 0,C 180,E1 -11934.044,E2 -11934.044} C_VEL
LIN {X 0,Y 383.095,Z 366.578,A -85,B 0,C 180,E1 -11935.443,E2 -11935.443} C_VEL
LIN {X 0,Y 386.809,Z 381.702,A -85,B 0,C 180,E1 -11938.644,E2 -11938.644} C_VEL
LIN {X 0,Y 389.575,Z 394,A -85,B 0,C 180,E1 -11941.077,E2 -11941.077} C_VEL
LIN {X 0,Y 390.856,Z 398.161,A -85,B 0,C 180,E1 -11941.251,E2 -11941.251} C_VEL
LIN {X 0,Y 397.237,Z 432.984,A -85,B 0,C 180,E1 -11942.374,E2 -11942.374} C_VEL
LIN {X 0,Y 394.632,Z 559.52,A -85,B 0,C 180,E1 -11944.696,E2 -11944.696} C_VEL
LIN {X 0,Y 393.85,Z 575.191,A -85,B 0,C 180,E1 -11945.172,E2 -11945.172} C_VEL
LIN {X 0,Y 392.798,Z 589.756,A -85,B 0,C 180,E1 -11945.814,E2 -11945.814} C_VEL
LIN {X 0,Y 391.634,Z 603.89,A -85,B 0,C 180,E1 -11946.645,E2 -11946.645} C_VEL
LIN {X 0,Y 390.271,Z 617.311,A -85,B 0,C 180,E1 -11947.64,E2 -11947.64} C_VEL
LIN {X 0,Y 388.876,Z 630.11,A -85,B 0,C 180,E1 -11948.81,E2 -11948.81} C_VEL
LIN {X 0,Y 387.411,Z 641.956,A -85,B 0,C 180,E1 -11950.114,E2 -11950.114} C_VEL
LIN {X 0,Y 386.256,Z 652.285,A -85,B 0,C 180,E1 -11951.467,E2 -11951.467} C_VEL
LIN {X 0,Y 385.044,Z 662.354,A -85,B 0,C 180,E1 -11953.02,E2 -11953.02} C_VEL
LIN {X 0,Y 383.929,Z 672.392,A -85,B 0,C 180,E1 -11954.879,E2 -11954.879} C_VEL
LIN {X 0,Y 383.008,Z 680.509,A -85,B 0,C 180,E1 -11956.688,E2 -11956.688} C_VEL
LIN {X 0,Y 382.518,Z 686.698,A -85,B 0,C 180,E1 -11958.34,E2 -11958.34} C_VEL
LIN {X 0,Y 381.974,Z 693.266,A -85,B 0,C 180,E1 -11960.468,E2 -11960.468} C_VEL
LIN {X 0,Y 381.73,Z 698.38,A -85,B 0,C 180,E1 -11962.595,E2 -11962.595} C_VEL
LIN {X 0,Y 381.584,Z 702.169,A -85,B 0,C 180,E1 -11964.716,E2 -11964.716} C_VEL
LIN {X 0,Y 381.537,Z 704.718,A -85,B 0,C 180,E1 -11966.832,E2 -11966.832} C_VEL
LIN {X 0,Y 381.636,Z 706.038,A -85,B 0,C 180,E1 -11968.945,E2 -11968.945} C_VEL
LIN {X 0,Y 381.634,Z 706.198,A -85,B 0,C 180,E1 -11971.055,E2 -11971.055} C_VEL
LIN {X 0,Y 381.533,Z 705.221,A -85,B 0,C 180,E1 -11973.168,E2 -11973.168} C_VEL
LIN {X 0,Y 381.574,Z 703.102,A -85,B 0,C 180,E1 -11975.284,E2 -11975.284} C_VEL
LIN {X 0,Y 381.727,Z 699.792,A -85,B 0,C 180,E1 -11977.405,E2 -11977.405} C_VEL
LIN {X 0,Y 382.018,Z 695.182,A -85,B 0,C 180,E1 -11979.531,E2 -11979.531} C_VEL
LIN {X 0,Y 382.628,Z 689.21,A -85,B 0,C 180,E1 -11981.657,E2 -11981.657} C_VEL
LIN {X 0,Y 383.372,Z 681.727,A -85,B 0,C 180,E1 -11983.787,E2 -11983.787} C_VEL
LIN {X 0,Y 384.497,Z 673.744,A -85,B 0,C 180,E1 -11985.641,E2 -11985.641} C_VEL
LIN {X 0,Y 385.831,Z 664.199,A -85,B 0,C 180,E1 -11987.491,E2 -11987.491} C_VEL
LIN {X 0,Y 387.322,Z 654.491,A -85,B 0,C 180,E1 -11989.063,E2 -11989.063} C_VEL
LIN {X 0,Y 388.92,Z 642.998,A -85,B 0,C 180,E1 -11990.633,E2 -11990.633} C_VEL
LIN {X 0,Y 390.716,Z 630.366,A -85,B 0,C 180,E1 -11992.055,E2 -11992.055} C_VEL
LIN {X 0,Y 392.44,Z 617.944,A -85,B 0,C 180,E1 -11993.203,E2 -11993.203} C_VEL
LIN {X 0,Y 394.008,Z 604.513,A -85,B 0,C 180,E1 -11994.221,E2 -11994.221} C_VEL
LIN {X 0,Y 395.394,Z 590.852,A -85,B 0,C 180,E1 -11995.042,E2 -11995.042} C_VEL
LIN {X 0,Y 396.566,Z 576.44,A -85,B 0,C 180,E1 -11995.699,E2 -11995.699} C_VEL
LIN {X 0,Y 397.556,Z 560.773,A -85,B 0,C 180,E1 -11996.193,E2 -11996.193} C_VEL
LIN {X 0,Y 399.171,Z 498.663,A -85,B 0,C 180,E1 -11997.366,E2 -11997.366} C_VEL
LIN {X 0,Y 400.687,Z 433.248,A -85,B 0,C 180,E1 -11998.582,E2 -11998.582} C_VEL
LIN {X 0,Y 396.59,Z 411.937,A -85,B 0,C 180,E1 -11999.392,E2 -11999.392} C_VEL
LIN {X 0,Y 394.164,Z 402.014,A -85,B 0,C 180,E1 -11999.826,E2 -11999.826} C_VEL
LIN {X 0,Y 390.232,Z 393.075,A -85,B 0,C 180,E1 -12000.42,E2 -12000.42} C_VEL
LIN {X 0,Y 386.954,Z 380.156,A -85,B 0,C 180,E1 -12003.336,E2 -12003.336} C_VEL
LIN {X 0,Y 383.462,Z 368.15,A -85,B 0,C 180,E1 -12006.253,E2 -12006.253} C_VEL
LIN {X 0,Y 383.009,Z 366.395,A -85,B 0,C 180,E1 -12006.742,E2 -12006.742} C_VEL
LIN {X 0,Y 382.973,Z 366.402,A -85,B 0,C 180,E1 -12009.963,E2 -12009.963} C_VEL
LIN {X 0,Y 383.004,Z 366.397,A -85,B 0,C 180,E1 -12012.779,E2 -12012.779} C_VEL
LIN {X 0,Y 382.994,Z 366.404,A -85,B 0,C 180,E1 -12015.789,E2 -12015.789} C_VEL
LIN {X 0,Y 382.96,Z 366.409,A -85,B 0,C 180,E1 -12018.801,E2 -12018.801} C_VEL
LIN {X 0,Y 382.991,Z 366.4,A -85,B 0,C 180,E1 -12022.098,E2 -12022.098} C_VEL
LIN {X 0,Y 383.017,Z 366.394,A -85,B 0,C 180,E1 -12025.332,E2 -12025.332} C_VEL
LIN {X 0,Y 383.009,Z 366.389,A -85,B 0,C 180,E1 -12027.851,E2 -12027.851} C_VEL
LIN {X 0,Y 382.985,Z 366.4,A -85,B 0,C 180,E1 -12031.503,E2 -12031.503} C_VEL
LIN {X 0,Y 383.028,Z 366.398,A -85,B 0,C 180,E1 -12035.038,E2 -12035.038} C_VEL
LIN {X 0,Y 382.999,Z 366.404,A -85,B 0,C 180,E1 -12038.47,E2 -12038.47} C_VEL
LIN {X 0,Y 383.061,Z 366.392,A -85,B 0,C 180,E1 -12041.827,E2 -12041.827} C_VEL
LIN {X 0,Y 383.109,Z 366.386,A -85,B 0,C 180,E1 -12045.119,E2 -12045.119} C_VEL
LIN {X 0,Y 383.097,Z 366.385,A -85,B 0,C 180,E1 -12048.358,E2 -12048.358} C_VEL
LIN {X 0,Y 383.216,Z 366.367,A -85,B 0,C 180,E1 -12052.028,E2 -12052.028} C_VEL
LIN {X 0,Y 383.183,Z 366.374,A -85,B 0,C 180,E1 -12054.739,E2 -12054.739} C_VEL
LIN {X 0,Y 383.384,Z 366.354,A -85,B 0,C 180,E1 -12057.899,E2 -12057.899} C_VEL
LIN {X 0,Y 383.302,Z 366.364,A -85,B 0,C 180,E1 -12061.051,E2 -12061.051} C_VEL
LIN {X 0,Y 383.211,Z 366.367,A -85,B 0,C 180,E1 -12063.154,E2 -12063.154} C_VEL
LIN {X 0,Y 383.225,Z 366.37,A -85,B 0,C 180,E1 -12066.534,E2 -12066.534} C_VEL
LIN {X 0,Y 383.145,Z 366.382,A -85,B 0,C 180,E1 -12069.503,E2 -12069.503} C_VEL
LIN {X 0,Y 383.128,Z 366.384,A -85,B 0,C 180,E1 -12073.537,E2 -12073.537} C_VEL
LIN {X 0,Y 383.097,Z 366.385,A -85,B 0,C 180,E1 -12077.455,E2 -12077.455} C_VEL
LIN {X 0,Y 383.031,Z 366.378,A -85,B 0,C 180,E1 -12080.647,E2 -12080.647} C_VEL
LIN {X 0,Y 383.013,Z 366.398,A -85,B 0,C 180,E1 -12083.809,E2 -12083.809} C_VEL
LIN {X 0,Y 383.02,Z 366.395,A -85,B 0,C 180,E1 -12087.305,E2 -12087.305} C_VEL
LIN {X 0,Y 382.985,Z 366.387,A -85,B 0,C 180,E1 -12090.919,E2 -12090.919} C_VEL
LIN {X 0,Y 383.015,Z 366.389,A -85,B 0,C 180,E1 -12094.669,E2 -12094.669} C_VEL
LIN {X 0,Y 382.995,Z 366.403,A -85,B 0,C 180,E1 -12097.903,E2 -12097.903} C_VEL
LIN {X 0,Y 382.964,Z 366.406,A -85,B 0,C 180,E1 -12101.351,E2 -12101.351} C_VEL
LIN {X 0,Y 382.998,Z 366.403,A -85,B 0,C 180,E1 -12104.303,E2 -12104.303} C_VEL
LIN {X 0,Y 383.036,Z 366.557,A -85,B 0,C 180,E1 -12107.217,E2 -12107.217} C_VEL
LIN {X 0,Y 385.092,Z 373.91,A -85,B 0,C 180,E1 -12109.149,E2 -12109.149} C_VEL
LIN {X 0,Y 395.083,Z 393.416,A -85,B 0,C 180,E1 -12110.547,E2 -12110.547} C_VEL
LIN {X 0,Y 401.208,Z 406.819,A -85,B 0,C 180,E1 -12111.387,E2 -12111.387} C_VEL
LIN {X 0,Y 398.408,Z 517.319,A -85,B 0,C 180,E1 -12113.423,E2 -12113.423} C_VEL
LIN {X 0,Y 397.851,Z 539.548,A -85,B 0,C 180,E1 -12113.874,E2 -12113.874} C_VEL
LIN {X 0,Y 397.019,Z 554.767,A -85,B 0,C 180,E1 -12114.368,E2 -12114.368} C_VEL
LIN {X 0,Y 395.931,Z 569.965,A -85,B 0,C 180,E1 -12115.085,E2 -12115.085} C_VEL
LIN {X 0,Y 394.648,Z 582.961,A -85,B 0,C 180,E1 -12115.878,E2 -12115.878} C_VEL
LIN {X 0,Y 393.239,Z 596.413,A -85,B 0,C 180,E1 -12116.922,E2 -12116.922} C_VEL
LIN {X 0,Y 391.549,Z 609.652,A -85,B 0,C 180,E1 -12118.18,E2 -12118.18} C_VEL
LIN {X 0,Y 389.846,Z 621.393,A -85,B 0,C 180,E1 -12119.534,E2 -12119.534} C_VEL
LIN {X 0,Y 388.274,Z 632.257,A -85,B 0,C 180,E1 -12121.04,E2 -12121.04} C_VEL
LIN {X 0,Y 386.789,Z 642.24,A -85,B 0,C 180,E1 -12122.691,E2 -12122.691} C_VEL
LIN {X 0,Y 385.243,Z 651.935,A -85,B 0,C 180,E1 -12124.614,E2 -12124.614} C_VEL
LIN {X 0,Y 384.074,Z 659.929,A -85,B 0,C 180,E1 -12126.547,E2 -12126.547} C_VEL
LIN {X 0,Y 383.128,Z 666.495,A -85,B 0,C 180,E1 -12128.477,E2 -12128.477} C_VEL
LIN {X 0,Y 382.424,Z 672.459,A -85,B 0,C 180,E1 -12130.683,E2 -12130.683} C_VEL
LIN {X 0,Y 382.012,Z 676.959,A -85,B 0,C 180,E1 -12132.881,E2 -12132.881} C_VEL
LIN {X 0,Y 381.652,Z 680.134,A -85,B 0,C 180,E1 -12135.06,E2 -12135.06} C_VEL
LIN {X 0,Y 381.603,Z 682.173,A -85,B 0,C 180,E1 -12137.452,E2 -12137.452} C_VEL
LIN {X 0,Y 381.482,Z 682.761,A -85,B 0,C 180,E1 -12139.384,E2 -12139.384} C_VEL
LIN {X 0,Y 381.473,Z 682.315,A -85,B 0,C 180,E1 -12141.525,E2 -12141.525} C_VEL
LIN {X 0,Y 381.709,Z 680.511,A -85,B 0,C 180,E1 -12143.857,E2 -12143.857} C_VEL
LIN {X 0,Y 381.757,Z 677.979,A -85,B 0,C 180,E1 -12145.777,E2 -12145.777} C_VEL
LIN {X 0,Y 382.017,Z 674.017,A -85,B 0,C 180,E1 -12147.891,E2 -12147.891} C_VEL
LIN {X 0,Y 382.345,Z 668.745,A -85,B 0,C 180,E1 -12150,E2 -12150} C_VEL
LIN {X 0,Y 383.072,Z 662.023,A -85,B 0,C 180,E1 -12152.103,E2 -12152.103} C_VEL
LIN {X 0,Y 383.894,Z 655.21,A -85,B 0,C 180,E1 -12153.835,E2 -12153.835} C_VEL
LIN {X 0,Y 383.62,Z 652.06,A -85,B 0,C 180,E1 -12154.58,E2 -12154.58} C_VEL
LIN {X 0,Y 381.459,Z 646.759,A -85,B 0,C 180,E1 -12155.795,E2 -12155.795} C_VEL
LIN {X 0,Y 379.394,Z 641.029,A -85,B 0,C 180,E1 -12156.974,E2 -12156.974} C_VEL
LIN {X 0,Y 379.264,Z 637.179,A -85,B 0,C 180,E1 -12157.652,E2 -12157.652} C_VEL
LIN {X 0,Y 380.683,Z 626.281,A -85,B 0,C 180,E1 -12159.296,E2 -12159.296} C_VEL
LIN {X 0,Y 382.11,Z 614.88,A -85,B 0,C 180,E1 -12160.733,E2 -12160.733} C_VEL
LIN {X 0,Y 383.501,Z 602.51,A -85,B 0,C 180,E1 -12162.032,E2 -12162.032} C_VEL
LIN {X 0,Y 384.958,Z 588.942,A -85,B 0,C 180,E1 -12163.192,E2 -12163.192} C_VEL
LIN {X 0,Y 386.167,Z 574.876,A -85,B 0,C 180,E1 -12164.156,E2 -12164.156} C_VEL
LIN {X 0,Y 387.239,Z 560.342,A -85,B 0,C 180,E1 -12164.921,E2 -12164.921} C_VEL
LIN {X 0,Y 387.989,Z 545.458,A -85,B 0,C 180,E1 -12165.497,E2 -12165.497} C_VEL
LIN {X 0,Y 388.579,Z 528.956,A -85,B 0,C 180,E1 -12165.895,E2 -12165.895} C_VEL
LIN {X 0,Y 391.135,Z 405.99,A -85,B 0,C 180,E1 -12168.172,E2 -12168.172} C_VEL
LIN {X 0,Y 381.46,Z 382.554,A -85,B 0,C 180,E1 -12169.346,E2 -12169.346} C_VEL
LIN {X 0,Y 377.5,Z 373.297,A -85,B 0,C 180,E1 -12169.872,E2 -12169.872} C_VEL
LIN {X 0,Y 375.957,Z 367.272,A -85,B 0,C 180,E1 -12171.378,E2 -12171.378} C_VEL
LIN {X 0,Y 375.94,Z 367.281,A -85,B 0,C 180,E1 -12174.285,E2 -12174.285} C_VEL
LIN {X 0,Y 375.924,Z 367.282,A -85,B 0,C 180,E1 -12176.66,E2 -12176.66} C_VEL
LIN {X 0,Y 375.92,Z 367.281,A -85,B 0,C 180,E1 -12179.084,E2 -12179.084} C_VEL
LIN {X 0,Y 375.962,Z 367.277,A -85,B 0,C 180,E1 -12181.562,E2 -12181.562} C_VEL
LIN {X 0,Y 375.96,Z 367.275,A -85,B 0,C 180,E1 -12185.415,E2 -12185.415} C_VEL
LIN {X 0,Y 375.938,Z 367.28,A -85,B 0,C 180,E1 -12188.262,E2 -12188.262} C_VEL
LIN {X 0,Y 375.92,Z 367.276,A -85,B 0,C 180,E1 -12191.597,E2 -12191.597} C_VEL
LIN {X 0,Y 375.929,Z 367.277,A -85,B 0,C 180,E1 -12194.731,E2 -12194.731} C_VEL
LIN {X 0,Y 375.929,Z 367.279,A -85,B 0,C 180,E1 -12197.698,E2 -12197.698} C_VEL
LIN {X 0,Y 375.937,Z 367.276,A -85,B 0,C 180,E1 -12200.533,E2 -12200.533} C_VEL
LIN {X 0,Y 375.961,Z 367.282,A -85,B 0,C 180,E1 -12203.497,E2 -12203.497} C_VEL
LIN {X 0,Y 375.96,Z 367.273,A -85,B 0,C 180,E1 -12205.888,E2 -12205.888} C_VEL
LIN {X 0,Y 375.965,Z 367.276,A -85,B 0,C 180,E1 -12209.687,E2 -12209.687} C_VEL
LIN {X 0,Y 375.921,Z 367.258,A -85,B 0,C 180,E1 -12212.135,E2 -12212.135} C_VEL
LIN {X 0,Y 375.938,Z 367.245,A -85,B 0,C 180,E1 -12214.533,E2 -12214.533} C_VEL
LIN {X 0,Y 375.977,Z 367.264,A -85,B 0,C 180,E1 -12216.886,E2 -12216.886} C_VEL
LIN {X 0,Y 376.002,Z 367.27,A -85,B 0,C 180,E1 -12220.339,E2 -12220.339} C_VEL
LIN {X 0,Y 376.029,Z 367.264,A -85,B 0,C 180,E1 -12223.718,E2 -12223.718} C_VEL
LIN {X 0,Y 376.106,Z 367.256,A -85,B 0,C 180,E1 -12227.042,E2 -12227.042} C_VEL
LIN {X 0,Y 376.115,Z 367.254,A -85,B 0,C 180,E1 -12230.318,E2 -12230.318} C_VEL
LIN {X 0,Y 376.196,Z 367.242,A -85,B 0,C 180,E1 -12233.564,E2 -12233.564} C_VEL
LIN {X 0,Y 376.34,Z 367.232,A -85,B 0,C 180,E1 -12237.859,E2 -12237.859} C_VEL
LIN {X 0,Y 376.236,Z 367.234,A -85,B 0,C 180,E1 -12241.07,E2 -12241.07} C_VEL
LIN {X 0,Y 376.346,Z 367.221,A -85,B 0,C 180,E1 -12242.14,E2 -12242.14} C_VEL
LIN {X 0,Y 376.2,Z 367.243,A -85,B 0,C 180,E1 -12246.435,E2 -12246.435} C_VEL
LIN {X 0,Y 376.115,Z 367.259,A -85,B 0,C 180,E1 -12249.681,E2 -12249.681} C_VEL
LIN {X 0,Y 376.091,Z 367.255,A -85,B 0,C 180,E1 -12253.657,E2 -12253.657} C_VEL
LIN {X 0,Y 376.013,Z 367.264,A -85,B 0,C 180,E1 -12257.591,E2 -12257.591} C_VEL
LIN {X 0,Y 375.979,Z 367.271,A -85,B 0,C 180,E1 -12260.832,E2 -12260.832} C_VEL
LIN {X 0,Y 375.972,Z 367.274,A -85,B 0,C 180,E1 -12264.283,E2 -12264.283} C_VEL
LIN {X 0,Y 375.928,Z 367.284,A -85,B 0,C 180,E1 -12267.864,E2 -12267.864} C_VEL
LIN {X 0,Y 375.958,Z 367.282,A -85,B 0,C 180,E1 -12271.562,E2 -12271.562} C_VEL
LIN {X 0,Y 375.956,Z 367.279,A -85,B 0,C 180,E1 -12275.415,E2 -12275.415} C_VEL
LIN {X 0,Y 375.933,Z 367.276,A -85,B 0,C 180,E1 -12278.262,E2 -12278.262} C_VEL
LIN {X 0,Y 375.916,Z 367.286,A -85,B 0,C 180,E1 -12281.597,E2 -12281.597} C_VEL
LIN {X 0,Y 375.924,Z 367.282,A -85,B 0,C 180,E1 -12284.731,E2 -12284.731} C_VEL
LIN {X 0,Y 375.924,Z 367.286,A -85,B 0,C 180,E1 -12287.698,E2 -12287.698} C_VEL
LIN {X 0,Y 375.933,Z 367.285,A -85,B 0,C 180,E1 -12290.534,E2 -12290.534} C_VEL
LIN {X 0,Y 375.961,Z 367.281,A -85,B 0,C 180,E1 -12293.496,E2 -12293.496} C_VEL
LIN {X 0,Y 376.022,Z 367.456,A -85,B 0,C 180,E1 -12295.006,E2 -12295.006} C_VEL
LIN {X 0,Y 379.843,Z 382.793,A -85,B 0,C 180,E1 -12298.332,E2 -12298.332} C_VEL
LIN {X 0,Y 382.249,Z 393.505,A -85,B 0,C 180,E1 -12300.537,E2 -12300.537} C_VEL
LIN {X 0,Y 384.617,Z 400.116,A -85,B 0,C 180,E1 -12300.846,E2 -12300.846} C_VEL
LIN {X 0,Y 390.721,Z 433.338,A -85,B 0,C 180,E1 -12301.944,E2 -12301.944} C_VEL
LIN {X 0,Y 388.063,Z 559.868,A -85,B 0,C 180,E1 -12304.309,E2 -12304.309} C_VEL
LIN {X 0,Y 387.266,Z 575.325,A -85,B 0,C 180,E1 -12304.792,E2 -12304.792} C_VEL
LIN {X 0,Y 386.147,Z 590.268,A -85,B 0,C 180,E1 -12305.467,E2 -12305.467} C_VEL
LIN {X 0,Y 384.926,Z 604.33,A -85,B 0,C 180,E1 -12306.317,E2 -12306.317} C_VEL
LIN {X 0,Y 383.447,Z 618.055,A -85,B 0,C 180,E1 -12307.362,E2 -12307.362} C_VEL
LIN {X 0,Y 382.038,Z 630.681,A -85,B 0,C 180,E1 -12308.554,E2 -12308.554} C_VEL
LIN {X 0,Y 380.515,Z 642.395,A -85,B 0,C 180,E1 -12309.879,E2 -12309.879} C_VEL
LIN {X 0,Y 379.214,Z 653.64,A -85,B 0,C 180,E1 -12311.409,E2 -12311.409} C_VEL
LIN {X 0,Y 377.974,Z 663.355,A -85,B 0,C 180,E1 -12312.971,E2 -12312.971} C_VEL
LIN {X 0,Y 376.826,Z 673.185,A -85,B 0,C 180,E1 -12314.864,E2 -12314.864} C_VEL
LIN {X 0,Y 375.942,Z 680.703,A -85,B 0,C 180,E1 -12316.587,E2 -12316.587} C_VEL
LIN {X 0,Y 375.337,Z 688.143,A -85,B 0,C 180,E1 -12318.661,E2 -12318.661} C_VEL
LIN {X 0,Y 374.828,Z 694.358,A -85,B 0,C 180,E1 -12320.829,E2 -12320.829} C_VEL
LIN {X 0,Y 374.627,Z 699.145,A -85,B 0,C 180,E1 -12322.996,E2 -12322.996} C_VEL
LIN {X 0,Y 374.5,Z 701.883,A -85,B 0,C 180,E1 -12324.616,E2 -12324.616} C_VEL
LIN {X 0,Y 374.451,Z 704.456,A -85,B 0,C 180,E1 -12326.772,E2 -12326.772} C_VEL
LIN {X 0,Y 374.537,Z 705.797,A -85,B 0,C 180,E1 -12328.925,E2 -12328.925} C_VEL
LIN {X 0,Y 374.535,Z 705.986,A -85,B 0,C 180,E1 -12331.075,E2 -12331.075} C_VEL
LIN {X 0,Y 374.447,Z 705.038,A -85,B 0,C 180,E1 -12333.228,E2 -12333.228} C_VEL
LIN {X 0,Y 374.491,Z 702.948,A -85,B 0,C 180,E1 -12335.384,E2 -12335.384} C_VEL
LIN {X 0,Y 374.652,Z 699.658,A -85,B 0,C 180,E1 -12337.545,E2 -12337.545} C_VEL
LIN {X 0,Y 374.971,Z 695.077,A -85,B 0,C 180,E1 -12339.711,E2 -12339.711} C_VEL
LIN {X 0,Y 375.621,Z 689.141,A -85,B 0,C 180,E1 -12341.877,E2 -12341.877} C_VEL
LIN {X 0,Y 376.439,Z 681.699,A -85,B 0,C 180,E1 -12344.046,E2 -12344.046} C_VEL
LIN {X 0,Y 377.611,Z 673.763,A -85,B 0,C 180,E1 -12345.934,E2 -12345.934} C_VEL
LIN {X 0,Y 379.032,Z 664.268,A -85,B 0,C 180,E1 -12347.815,E2 -12347.815} C_VEL
LIN {X 0,Y 380.719,Z 653.704,A -85,B 0,C 180,E1 -12349.552,E2 -12349.552} C_VEL
LIN {X 0,Y 382.428,Z 642.143,A -85,B 0,C 180,E1 -12351.14,E2 -12351.14} C_VEL
LIN {X 0,Y 384.336,Z 629.383,A -85,B 0,C 180,E1 -12352.582,E2 -12352.582} C_VEL
LIN {X 0,Y 386.347,Z 615.224,A -85,B 0,C 180,E1 -12353.875,E2 -12353.875} C_VEL
LIN {X 0,Y 387.992,Z 601.536,A -85,B 0,C 180,E1 -12354.88,E2 -12354.88} C_VEL
LIN {X 0,Y 389.337,Z 587.923,A -85,B 0,C 180,E1 -12355.673,E2 -12355.673} C_VEL
LIN {X 0,Y 390.5,Z 574.327,A -85,B 0,C 180,E1 -12356.271,E2 -12356.271} C_VEL
LIN {X 0,Y 391.477,Z 558.869,A -85,B 0,C 180,E1 -12356.74,E2 -12356.74} C_VEL
LIN {X 0,Y 394.627,Z 434.472,A -85,B 0,C 180,E1 -12359.095,E2 -12359.095} C_VEL
LIN {X 0,Y 390.812,Z 414.382,A -85,B 0,C 180,E1 -12359.876,E2 -12359.876} C_VEL
LIN {X 0,Y 388.619,Z 405.159,A -85,B 0,C 180,E1 -12360.285,E2 -12360.285} C_VEL
LIN {X 0,Y 382.967,Z 392.834,A -85,B 0,C 180,E1 -12361.138,E2 -12361.138} C_VEL
LIN {X 0,Y 379.361,Z 378.883,A -85,B 0,C 180,E1 -12364.404,E2 -12364.404} C_VEL
LIN {X 0,Y 375.957,Z 367.278,A -85,B 0,C 180,E1 -12367.349,E2 -12367.349} C_VEL
LIN {X 0,Y 375.913,Z 367.281,A -85,B 0,C 180,E1 -12370.871,E2 -12370.871} C_VEL
LIN {X 0,Y 375.927,Z 367.284,A -85,B 0,C 180,E1 -12373.766,E2 -12373.766} C_VEL
LIN {X 0,Y 375.933,Z 367.284,A -85,B 0,C 180,E1 -12376.811,E2 -12376.811} C_VEL
LIN {X 0,Y 375.933,Z 367.281,A -85,B 0,C 180,E1 -12380.534,E2 -12380.534} C_VEL
LIN {X 0,Y 375.961,Z 367.26,A -85,B 0,C 180,E1 -12383.496,E2 -12383.496} C_VEL
LIN {X 0,Y 375.96,Z 367.275,A -85,B 0,C 180,E1 -12385.889,E2 -12385.889} C_VEL
LIN {X 0,Y 375.962,Z 367.255,A -85,B 0,C 180,E1 -12389.688,E2 -12389.688} C_VEL
LIN {X 0,Y 375.933,Z 367.276,A -85,B 0,C 180,E1 -12393.342,E2 -12393.342} C_VEL
LIN {X 0,Y 375.979,Z 367.27,A -85,B 0,C 180,E1 -12396.888,E2 -12396.888} C_VEL
LIN {X 0,Y 375.997,Z 367.27,A -85,B 0,C 180,E1 -12400.34,E2 -12400.34} C_VEL
LIN {X 0,Y 376.028,Z 367.266,A -85,B 0,C 180,E1 -12403.719,E2 -12403.719} C_VEL
LIN {X 0,Y 376.104,Z 367.255,A -85,B 0,C 180,E1 -12407.043,E2 -12407.043} C_VEL
LIN {X 0,Y 376.114,Z 367.26,A -85,B 0,C 180,E1 -12410.319,E2 -12410.319} C_VEL
LIN {X 0,Y 376.202,Z 367.247,A -85,B 0,C 180,E1 -12413.565,E2 -12413.565} C_VEL
LIN {X 0,Y 376.35,Z 367.23,A -85,B 0,C 180,E1 -12417.86,E2 -12417.86} C_VEL
LIN {X 0,Y 376.27,Z 367.24,A -85,B 0,C 180,E1 -12421.071,E2 -12421.071} C_VEL
LIN {X 0,Y 376.344,Z 367.233,A -85,B 0,C 180,E1 -12422.141,E2 -12422.141} C_VEL
LIN {X 0,Y 376.194,Z 367.246,A -85,B 0,C 180,E1 -12426.519,E2 -12426.519} C_VEL
LIN {X 0,Y 376.115,Z 367.258,A -85,B 0,C 180,E1 -12429.682,E2 -12429.682} C_VEL
LIN {X 0,Y 376.092,Z 367.26,A -85,B 0,C 180,E1 -12433.658,E2 -12433.658} C_VEL
LIN {X 0,Y 376.046,Z 367.264,A -85,B 0,C 180,E1 -12437.607,E2 -12437.607} C_VEL
LIN {X 0,Y 375.981,Z 367.258,A -85,B 0,C 180,E1 -12440.833,E2 -12440.833} C_VEL
LIN {X 0,Y 375.962,Z 367.268,A -85,B 0,C 180,E1 -12444.284,E2 -12444.284} C_VEL
LIN {X 0,Y 375.96,Z 367.276,A -85,B 0,C 180,E1 -12447.862,E2 -12447.862} C_VEL
LIN {X 0,Y 375.96,Z 367.264,A -85,B 0,C 180,E1 -12451.562,E2 -12451.562} C_VEL
LIN {X 0,Y 375.953,Z 367.264,A -85,B 0,C 180,E1 -12455.417,E2 -12455.417} C_VEL
LIN {X 0,Y 375.937,Z 367.278,A -85,B 0,C 180,E1 -12458.263,E2 -12458.263} C_VEL
LIN {X 0,Y 375.92,Z 367.282,A -85,B 0,C 180,E1 -12461.598,E2 -12461.598} C_VEL
LIN {X 0,Y 375.929,Z 367.279,A -85,B 0,C 180,E1 -12464.732,E2 -12464.732} C_VEL
LIN {X 0,Y 375.992,Z 367.412,A -85,B 0,C 180,E1 -12466.576,E2 -12466.576} C_VEL
LIN {X 0,Y 377.927,Z 374.314,A -85,B 0,C 180,E1 -12468.411,E2 -12468.411} C_VEL
LIN {X 0,Y 387.831,Z 392.993,A -85,B 0,C 180,E1 -12469.843,E2 -12469.843} C_VEL
LIN {X 0,Y 395.207,Z 409.027,A -85,B 0,C 180,E1 -12470.89,E2 -12470.89} C_VEL
LIN {X 0,Y 392.083,Z 523.307,A -85,B 0,C 180,E1 -12473.015,E2 -12473.015} C_VEL
LIN {X 0,Y 391.584,Z 542.287,A -85,B 0,C 180,E1 -12473.442,E2 -12473.442} C_VEL
LIN {X 0,Y 390.644,Z 557.337,A -85,B 0,C 180,E1 -12473.969,E2 -12473.969} C_VEL
LIN {X 0,Y 389.437,Z 572.465,A -85,B 0,C 180,E1 -12474.726,E2 -12474.726} C_VEL
LIN {X 0,Y 388.157,Z 585.093,A -85,B 0,C 180,E1 -12475.541,E2 -12475.541} C_VEL
LIN {X 0,Y 386.547,Z 598.958,A -85,B 0,C 180,E1 -12476.665,E2 -12476.665} C_VEL
LIN {X 0,Y 384.904,Z 611.16,A -85,B 0,C 180,E1 -12477.873,E2 -12477.873} C_VEL
LIN {X 0,Y 383.097,Z 623.072,A -85,B 0,C 180,E1 -12479.295,E2 -12479.295} C_VEL
LIN {X 0,Y 381.491,Z 633.394,A -85,B 0,C 180,E1 -12480.778,E2 -12480.778} C_VEL
LIN {X 0,Y 379.735,Z 644.401,A -85,B 0,C 180,E1 -12482.67,E2 -12482.67} C_VEL
LIN {X 0,Y 378.183,Z 654.039,A -85,B 0,C 180,E1 -12484.696,E2 -12484.696} C_VEL
LIN {X 0,Y 377.109,Z 660.761,A -85,B 0,C 180,E1 -12486.408,E2 -12486.408} C_VEL
LIN {X 0,Y 376.008,Z 667.945,A -85,B 0,C 180,E1 -12488.625,E2 -12488.625} C_VEL
LIN {X 0,Y 375.323,Z 673.62,A -85,B 0,C 180,E1 -12490.871,E2 -12490.871} C_VEL
LIN {X 0,Y 374.927,Z 677.582,A -85,B 0,C 180,E1 -12492.941,E2 -12492.941} C_VEL
LIN {X 0,Y 374.595,Z 680.2,A -85,B 0,C 180,E1 -12494.772,E2 -12494.772} C_VEL
LIN {X 0,Y 374.501,Z 682.173,A -85,B 0,C 180,E1 -12496.986,E2 -12496.986} C_VEL
LIN {X 0,Y 374.402,Z 682.961,A -85,B 0,C 180,E1 -12499.181,E2 -12499.181} C_VEL
LIN {X 0,Y 374.381,Z 682.597,A -85,B 0,C 180,E1 -12501.363,E2 -12501.363} C_VEL
LIN {X 0,Y 374.555,Z 681.088,A -85,B 0,C 180,E1 -12503.536,E2 -12503.536} C_VEL
LIN {X 0,Y 374.673,Z 678.426,A -85,B 0,C 180,E1 -12505.697,E2 -12505.697} C_VEL
LIN {X 0,Y 374.941,Z 674.524,A -85,B 0,C 180,E1 -12507.852,E2 -12507.852} C_VEL
LIN {X 0,Y 375.268,Z 669.323,A -85,B 0,C 180,E1 -12510,E2 -12510} C_VEL
LIN {X 0,Y 375.998,Z 662.698,A -85,B 0,C 180,E1 -12512.142,E2 -12512.142} C_VEL
LIN {X 0,Y 377.034,Z 654.46,A -85,B 0,C 180,E1 -12514.276,E2 -12514.276} C_VEL
LIN {X 0,Y 378.173,Z 645.681,A -85,B 0,C 180,E1 -12516.134,E2 -12516.134} C_VEL
LIN {X 0,Y 379.264,Z 637.179,A -85,B 0,C 180,E1 -12517.652,E2 -12517.652} C_VEL
LIN {X 0,Y 379.172,Z 633.239,A -85,B 0,C 180,E1 -12518.315,E2 -12518.315} C_VEL
LIN {X 0,Y 377.31,Z 626.706,A -85,B 0,C 180,E1 -12519.414,E2 -12519.414} C_VEL
LIN {X 0,Y 375.442,Z 619.825,A -85,B 0,C 180,E1 -12520.465,E2 -12520.465} C_VEL
LIN {X 0,Y 375.331,Z 615.285,A -85,B 0,C 180,E1 -12521.042,E2 -12521.042} C_VEL
LIN {X 0,Y 376.816,Z 602.709,A -85,B 0,C 180,E1 -12522.386,E2 -12522.386} C_VEL
LIN {X 0,Y 378.32,Z 589.137,A -85,B 0,C 180,E1 -12523.564,E2 -12523.564} C_VEL
LIN {X 0,Y 379.579,Z 575.054,A -85,B 0,C 180,E1 -12524.543,E2 -12524.543} C_VEL
LIN {X 0,Y 380.671,Z 560.507,A -85,B 0,C 180,E1 -12525.322,E2 -12525.322} C_VEL
LIN {X 0,Y 381.465,Z 545.577,A -85,B 0,C 180,E1 -12525.906,E2 -12525.906} C_VEL
LIN {X 0,Y 382.031,Z 530.031,A -85,B 0,C 180,E1 -12526.293,E2 -12526.293} C_VEL
LIN {X 0,Y 384.756,Z 408.092,A -85,B 0,C 180,E1 -12528.579,E2 -12528.579} C_VEL
LIN {X 0,Y 376.884,Z 388.531,A -85,B 0,C 180,E1 -12529.566,E2 -12529.566} C_VEL
LIN {X 0,Y 370.29,Z 373.627,A -85,B 0,C 180,E1 -12530.412,E2 -12530.412} C_VEL
LIN {X 0,Y 368.939,Z 368.15,A -85,B 0,C 180,E1 -12531.805,E2 -12531.805} C_VEL
LIN {X 0,Y 368.891,Z 368.158,A -85,B 0,C 180,E1 -12534.78,E2 -12534.78} C_VEL
LIN {X 0,Y 368.915,Z 368.155,A -85,B 0,C 180,E1 -12538.442,E2 -12538.442} C_VEL
LIN {X 0,Y 368.915,Z 368.155,A -85,B 0,C 180,E1 -12540.987,E2 -12540.987} C_VEL
LIN {X 0,Y 368.94,Z 368.152,A -85,B 0,C 180,E1 -12544.853,E2 -12544.853} C_VEL
LIN {X 0,Y 368.879,Z 368.159,A -85,B 0,C 180,E1 -12548.633,E2 -12548.633} C_VEL
LIN {X 0,Y 368.874,Z 368.16,A -85,B 0,C 180,E1 -12552.007,E2 -12552.007} C_VEL
LIN {X 0,Y 368.882,Z 368.151,A -85,B 0,C 180,E1 -12555.175,E2 -12555.175} C_VEL
LIN {X 0,Y 368.873,Z 368.16,A -85,B 0,C 180,E1 -12558.175,E2 -12558.175} C_VEL
LIN {X 0,Y 368.879,Z 368.155,A -85,B 0,C 180,E1 -12561.366,E2 -12561.366} C_VEL
LIN {X 0,Y 368.934,Z 368.152,A -85,B 0,C 180,E1 -12565.145,E2 -12565.145} C_VEL
LIN {X 0,Y 368.916,Z 368.157,A -85,B 0,C 180,E1 -12569.045,E2 -12569.045} C_VEL
LIN {X 0,Y 368.91,Z 368.136,A -85,B 0,C 180,E1 -12571.557,E2 -12571.557} C_VEL
LIN {X 0,Y 368.889,Z 368.127,A -85,B 0,C 180,E1 -12575.219,E2 -12575.219} C_VEL
LIN {X 0,Y 368.924,Z 368.149,A -85,B 0,C 180,E1 -12577.604,E2 -12577.604} C_VEL
LIN {X 0,Y 368.958,Z 368.149,A -85,B 0,C 180,E1 -12581.105,E2 -12581.105} C_VEL
LIN {X 0,Y 369,Z 368.141,A -85,B 0,C 180,E1 -12584.535,E2 -12584.535} C_VEL
LIN {X 0,Y 369.007,Z 368.131,A -85,B 0,C 180,E1 -12587.906,E2 -12587.906} C_VEL
LIN {X 0,Y 369.093,Z 368.131,A -85,B 0,C 180,E1 -12591.237,E2 -12591.237} C_VEL
LIN {X 0,Y 369.119,Z 368.116,A -85,B 0,C 180,E1 -12594.537,E2 -12594.537} C_VEL
LIN {X 0,Y 369.304,Z 368.109,A -85,B 0,C 180,E1 -12597.818,E2 -12597.818} C_VEL
LIN {X 0,Y 369.207,Z 368.109,A -85,B 0,C 180,E1 -12601.09,E2 -12601.09} C_VEL
LIN {X 0,Y 369.31,Z 368.097,A -85,B 0,C 180,E1 -12602.181,E2 -12602.181} C_VEL
LIN {X 0,Y 369.161,Z 368.119,A -85,B 0,C 180,E1 -12606.559,E2 -12606.559} C_VEL
LIN {X 0,Y 369.065,Z 368.138,A -85,B 0,C 180,E1 -12609.868,E2 -12609.868} C_VEL
LIN {X 0,Y 369.039,Z 368.134,A -85,B 0,C 180,E1 -12613.772,E2 -12613.772} C_VEL
LIN {X 0,Y 368.978,Z 368.14,A -85,B 0,C 180,E1 -12617.756,E2 -12617.756} C_VEL
LIN {X 0,Y 368.93,Z 368.152,A -85,B 0,C 180,E1 -12621.219,E2 -12621.219} C_VEL
LIN {X 0,Y 368.926,Z 368.151,A -85,B 0,C 180,E1 -12624.777,E2 -12624.777} C_VEL
LIN {X 0,Y 368.897,Z 368.156,A -85,B 0,C 180,E1 -12628.793,E2 -12628.793} C_VEL
LIN {X 0,Y 368.898,Z 368.155,A -85,B 0,C 180,E1 -12632.238,E2 -12632.238} C_VEL
LIN {X 0,Y 368.928,Z 368.154,A -85,B 0,C 180,E1 -12635.001,E2 -12635.001} C_VEL
LIN {X 0,Y 368.875,Z 368.154,A -85,B 0,C 180,E1 -12638.633,E2 -12638.633} C_VEL
LIN {X 0,Y 368.869,Z 368.161,A -85,B 0,C 180,E1 -12642.007,E2 -12642.007} C_VEL
LIN {X 0,Y 368.877,Z 368.161,A -85,B 0,C 180,E1 -12645.175,E2 -12645.175} C_VEL
LIN {X 0,Y 368.868,Z 368.165,A -85,B 0,C 180,E1 -12648.175,E2 -12648.175} C_VEL
LIN {X 0,Y 368.875,Z 368.164,A -85,B 0,C 180,E1 -12651.366,E2 -12651.366} C_VEL
LIN {X 0,Y 368.948,Z 368.308,A -85,B 0,C 180,E1 -12654.547,E2 -12654.547} C_VEL
LIN {X 0,Y 372.219,Z 381.297,A -85,B 0,C 180,E1 -12657.445,E2 -12657.445} C_VEL
LIN {X 0,Y 375.039,Z 393.399,A -85,B 0,C 180,E1 -12659.994,E2 -12659.994} C_VEL
LIN {X 0,Y 378.446,Z 402.418,A -85,B 0,C 180,E1 -12660.44,E2 -12660.44} C_VEL
LIN {X 0,Y 384.288,Z 434.294,A -85,B 0,C 180,E1 -12661.519,E2 -12661.519} C_VEL
LIN {X 0,Y 381.5,Z 560.088,A -85,B 0,C 180,E1 -12663.907,E2 -12663.907} C_VEL
LIN {X 0,Y 380.6,Z 576.179,A -85,B 0,C 180,E1 -12664.429,E2 -12664.429} C_VEL
LIN {X 0,Y 379.482,Z 590.875,A -85,B 0,C 180,E1 -12665.117,E2 -12665.117} C_VEL
LIN {X 0,Y 378.161,Z 605.258,A -85,B 0,C 180,E1 -12666.012,E2 -12666.012} C_VEL
LIN {X 0,Y 376.658,Z 618.777,A -85,B 0,C 180,E1 -12667.076,E2 -12667.076} C_VEL
LIN {X 0,Y 375.002,Z 632.518,A -85,B 0,C 180,E1 -12668.42,E2 -12668.42} C_VEL
LIN {X 0,Y 373.426,Z 644.977,A -85,B 0,C 180,E1 -12669.911,E2 -12669.911} C_VEL
LIN {X 0,Y 372.027,Z 656.329,A -85,B 0,C 180,E1 -12671.553,E2 -12671.553} C_VEL
LIN {X 0,Y 370.542,Z 667.317,A -85,B 0,C 180,E1 -12673.471,E2 -12673.471} C_VEL
LIN {X 0,Y 369.431,Z 676.451,A -85,B 0,C 180,E1 -12675.4,E2 -12675.4} C_VEL
LIN {X 0,Y 368.649,Z 684.02,A -85,B 0,C 180,E1 -12677.336,E2 -12677.336} C_VEL
LIN {X 0,Y 367.945,Z 691.06,A -85,B 0,C 180,E1 -12679.545,E2 -12679.545} C_VEL
LIN {X 0,Y 367.627,Z 696.583,A -85,B 0,C 180,E1 -12681.756,E2 -12681.756} C_VEL
LIN {X 0,Y 367.476,Z 700.779,A -85,B 0,C 180,E1 -12683.988,E2 -12683.988} C_VEL
LIN {X 0,Y 367.423,Z 703.053,A -85,B 0,C 180,E1 -12685.612,E2 -12685.612} C_VEL
LIN {X 0,Y 367.392,Z 705.016,A -85,B 0,C 180,E1 -12687.807,E2 -12687.807} C_VEL
LIN {X 0,Y 367.469,Z 705.808,A -85,B 0,C 180,E1 -12690,E2 -12690} C_VEL
LIN {X 0,Y 367.374,Z 705.456,A -85,B 0,C 180,E1 -12692.193,E2 -12692.193} C_VEL
LIN {X 0,Y 367.397,Z 703.971,A -85,B 0,C 180,E1 -12694.388,E2 -12694.388} C_VEL
LIN {X 0,Y 367.48,Z 701.32,A -85,B 0,C 180,E1 -12696.589,E2 -12696.589} C_VEL
LIN {X 0,Y 367.741,Z 697.411,A -85,B 0,C 180,E1 -12698.794,E2 -12698.794} C_VEL
LIN {X 0,Y 368.171,Z 692.203,A -85,B 0,C 180,E1 -12701.005,E2 -12701.005} C_VEL
LIN {X 0,Y 368.984,Z 685.576,A -85,B 0,C 180,E1 -12703.212,E2 -12703.212} C_VEL
LIN {X 0,Y 369.996,Z 678.468,A -85,B 0,C 180,E1 -12705.14,E2 -12705.14} C_VEL
LIN {X 0,Y 371.324,Z 669.959,A -85,B 0,C 180,E1 -12707.06,E2 -12707.06} C_VEL
LIN {X 0,Y 372.798,Z 661.367,A -85,B 0,C 180,E1 -12708.692,E2 -12708.692} C_VEL
LIN {X 0,Y 374.43,Z 651.061,A -85,B 0,C 180,E1 -12710.344,E2 -12710.344} C_VEL
LIN {X 0,Y 376.361,Z 639.177,A -85,B 0,C 180,E1 -12711.93,E2 -12711.93} C_VEL
LIN {X 0,Y 378.186,Z 627.142,A -85,B 0,C 180,E1 -12713.26,E2 -12713.26} C_VEL
LIN {X 0,Y 380.105,Z 614.106,A -85,B 0,C 180,E1 -12714.438,E2 -12714.438} C_VEL
LIN {X 0,Y 381.833,Z 599.829,A -85,B 0,C 180,E1 -12715.482,E2 -12715.482} C_VEL
LIN {X 0,Y 383.246,Z 586.23,A -85,B 0,C 180,E1 -12716.258,E2 -12716.258} C_VEL
LIN {X 0,Y 384.54,Z 571.125,A -85,B 0,C 180,E1 -12716.894,E2 -12716.894} C_VEL
LIN {X 0,Y 385.418,Z 556.737,A -85,B 0,C 180,E1 -12717.304,E2 -12717.304} C_VEL
LIN {X 0,Y 388.589,Z 435.836,A -85,B 0,C 180,E1 -12719.623,E2 -12719.623} C_VEL
LIN {X 0,Y 384.93,Z 416.102,A -85,B 0,C 180,E1 -12720.405,E2 -12720.405} C_VEL
LIN {X 0,Y 383.072,Z 408.263,A -85,B 0,C 180,E1 -12720.762,E2 -12720.762} C_VEL
LIN {X 0,Y 377.3,Z 396.052,A -85,B 0,C 180,E1 -12721.629,E2 -12721.629} C_VEL
LIN {X 0,Y 375.727,Z 392.586,A -85,B 0,C 180,E1 -12721.895,E2 -12721.895} C_VEL
LIN {X 0,Y 372.31,Z 379.628,A -85,B 0,C 180,E1 -12725.032,E2 -12725.032} C_VEL
LIN {X 0,Y 368.932,Z 368.15,A -85,B 0,C 180,E1 -12728.078,E2 -12728.078} C_VEL
LIN {X 0,Y 368.869,Z 368.151,A -85,B 0,C 180,E1 -12732.008,E2 -12732.008} C_VEL
LIN {X 0,Y 368.877,Z 368.162,A -85,B 0,C 180,E1 -12735.176,E2 -12735.176} C_VEL
LIN {X 0,Y 368.867,Z 368.161,A -85,B 0,C 180,E1 -12738.176,E2 -12738.176} C_VEL
LIN {X 0,Y 368.875,Z 368.16,A -85,B 0,C 180,E1 -12741.366,E2 -12741.366} C_VEL
LIN {X 0,Y 368.935,Z 368.145,A -85,B 0,C 180,E1 -12745.147,E2 -12745.147} C_VEL
LIN {X 0,Y 368.929,Z 368.128,A -85,B 0,C 180,E1 -12749.047,E2 -12749.047} C_VEL
LIN {X 0,Y 368.875,Z 368.158,A -85,B 0,C 180,E1 -12752.79,E2 -12752.79} C_VEL
LIN {X 0,Y 368.928,Z 368.154,A -85,B 0,C 180,E1 -12756.119,E2 -12756.119} C_VEL
LIN {X 0,Y 368.936,Z 368.151,A -85,B 0,C 180,E1 -12759.947,E2 -12759.947} C_VEL
LIN {X 0,Y 368.975,Z 368.144,A -85,B 0,C 180,E1 -12763.399,E2 -12763.399} C_VEL
LIN {X 0,Y 369.059,Z 368.134,A -85,B 0,C 180,E1 -12766.791,E2 -12766.791} C_VEL
LIN {X 0,Y 369.064,Z 368.139,A -85,B 0,C 180,E1 -12770.132,E2 -12770.132} C_VEL
LIN {X 0,Y 369.162,Z 368.124,A -85,B 0,C 180,E1 -12773.441,E2 -12773.441} C_VEL
LIN {X 0,Y 369.315,Z 368.106,A -85,B 0,C 180,E1 -12777.819,E2 -12777.819} C_VEL
LIN {X 0,Y 369.237,Z 368.116,A -85,B 0,C 180,E1 -12781.091,E2 -12781.091} C_VEL
LIN {X 0,Y 369.308,Z 368.109,A -85,B 0,C 180,E1 -12782.182,E2 -12782.182} C_VEL
LIN {X 0,Y 369.163,Z 368.121,A -85,B 0,C 180,E1 -12786.56,E2 -12786.56} C_VEL
LIN {X 0,Y 369.065,Z 368.137,A -85,B 0,C 180,E1 -12789.869,E2 -12789.869} C_VEL
LIN {X 0,Y 369.04,Z 368.139,A -85,B 0,C 180,E1 -12793.773,E2 -12793.773} C_VEL
LIN {X 0,Y 369.004,Z 368.14,A -85,B 0,C 180,E1 -12797.769,E2 -12797.769} C_VEL
LIN {X 0,Y 368.912,Z 368.145,A -85,B 0,C 180,E1 -12801.221,E2 -12801.221} C_VEL
LIN {X 0,Y 368.922,Z 368.152,A -85,B 0,C 180,E1 -12803.878,E2 -12803.878} C_VEL
LIN {X 0,Y 368.891,Z 368.151,A -85,B 0,C 180,E1 -12807.21,E2 -12807.21} C_VEL
LIN {X 0,Y 368.903,Z 368.152,A -85,B 0,C 180,E1 -12809.692,E2 -12809.692} C_VEL
LIN {X 0,Y 368.9,Z 368.16,A -85,B 0,C 180,E1 -12813.044,E2 -12813.044} C_VEL
LIN {X 0,Y 368.914,Z 368.144,A -85,B 0,C 180,E1 -12816.198,E2 -12816.198} C_VEL
LIN {X 0,Y 368.876,Z 368.15,A -85,B 0,C 180,E1 -12818.957,E2 -12818.957} C_VEL
LIN {X 0,Y 368.873,Z 368.155,A -85,B 0,C 180,E1 -12822.008,E2 -12822.008} C_VEL
LIN {X 0,Y 368.9,Z 368.153,A -85,B 0,C 180,E1 -12825.811,E2 -12825.811} C_VEL
LIN {X 0,Y 370.613,Z 374.34,A -85,B 0,C 180,E1 -12827.61,E2 -12827.61} C_VEL
LIN {X 0,Y 380.233,Z 392.158,A -85,B 0,C 180,E1 -12829.059,E2 -12829.059} C_VEL
LIN {X 0,Y 388.716,Z 409.986,A -85,B 0,C 180,E1 -12830.3,E2 -12830.3} C_VEL
LIN {X 0,Y 389.125,Z 410.889,A -85,B 0,C 180,E1 -12830.359,E2 -12830.359} C_VEL
LIN {X 0,Y 386.21,Z 516.309,A -85,B 0,C 180,E1 -12832.356,E2 -12832.356} C_VEL
LIN {X 0,Y 385.519,Z 540.238,A -85,B 0,C 180,E1 -12832.852,E2 -12832.852} C_VEL
LIN {X 0,Y 384.613,Z 555.487,A -85,B 0,C 180,E1 -12833.365,E2 -12833.365} C_VEL
LIN {X 0,Y 383.445,Z 570.411,A -85,B 0,C 180,E1 -12834.09,E2 -12834.09} C_VEL
LIN {X 0,Y 382.028,Z 583.482,A -85,B 0,C 180,E1 -12834.908,E2 -12834.908} C_VEL
LIN {X 0,Y 380.425,Z 597.411,A -85,B 0,C 180,E1 -12836.024,E2 -12836.024} C_VEL
LIN {X 0,Y 378.625,Z 610.208,A -85,B 0,C 180,E1 -12837.284,E2 -12837.284} C_VEL
LIN {X 0,Y 376.675,Z 622.56,A -85,B 0,C 180,E1 -12838.761,E2 -12838.761} C_VEL
LIN {X 0,Y 374.985,Z 632.701,A -85,B 0,C 180,E1 -12840.22,E2 -12840.22} C_VEL
LIN {X 0,Y 373.375,Z 642.678,A -85,B 0,C 180,E1 -12841.929,E2 -12841.929} C_VEL
LIN {X 0,Y 371.837,Z 651.101,A -85,B 0,C 180,E1 -12843.63,E2 -12843.63} C_VEL
LIN {X 0,Y 370.479,Z 659.163,A -85,B 0,C 180,E1 -12845.585,E2 -12845.585} C_VEL
LIN {X 0,Y 369.4,Z 666.102,A -85,B 0,C 180,E1 -12847.635,E2 -12847.635} C_VEL
LIN {X 0,Y 368.5,Z 672.258,A -85,B 0,C 180,E1 -12849.922,E2 -12849.922} C_VEL
LIN {X 0,Y 367.958,Z 676.931,A -85,B 0,C 180,E1 -12852.206,E2 -12852.206} C_VEL
LIN {X 0,Y 367.552,Z 680.238,A -85,B 0,C 180,E1 -12854.473,E2 -12854.473} C_VEL
LIN {X 0,Y 367.396,Z 682.292,A -85,B 0,C 180,E1 -12856.729,E2 -12856.729} C_VEL
LIN {X 0,Y 367.334,Z 683.16,A -85,B 0,C 180,E1 -12858.97,E2 -12858.97} C_VEL
LIN {X 0,Y 367.285,Z 682.878,A -85,B 0,C 180,E1 -12861.195,E2 -12861.195} C_VEL
LIN {X 0,Y 367.461,Z 681.449,A -85,B 0,C 180,E1 -12863.411,E2 -12863.411} C_VEL
LIN {X 0,Y 367.59,Z 678.854,A -85,B 0,C 180,E1 -12865.614,E2 -12865.614} C_VEL
LIN {X 0,Y 367.866,Z 675.009,A -85,B 0,C 180,E1 -12867.81,E2 -12867.81} C_VEL
LIN {X 0,Y 368.193,Z 669.896,A -85,B 0,C 180,E1 -12870,E2 -12870} C_VEL
LIN {X 0,Y 368.925,Z 663.367,A -85,B 0,C 180,E1 -12872.184,E2 -12872.184} C_VEL
LIN {X 0,Y 369.854,Z 656.335,A -85,B 0,C 180,E1 -12874.086,E2 -12874.086} C_VEL
LIN {X 0,Y 371.002,Z 647.903,A -85,B 0,C 180,E1 -12875.98,E2 -12875.98} C_VEL
LIN {X 0,Y 372.358,Z 637.786,A -85,B 0,C 180,E1 -12877.865,E2 -12877.865} C_VEL
LIN {X 0,Y 373.765,Z 627.453,A -85,B 0,C 180,E1 -12879.47,E2 -12879.47} C_VEL
LIN {X 0,Y 375.331,Z 615.285,A -85,B 0,C 180,E1 -12881.042,E2 -12881.042} C_VEL
LIN {X 0,Y 375.246,Z 610.679,A -85,B 0,C 180,E1 -12881.605,E2 -12881.605} C_VEL
LIN {X 0,Y 371.932,Z 596.84,A -85,B 0,C 180,E1 -12883.261,E2 -12883.261} C_VEL
LIN {X 0,Y 371.51,Z 591.854,A -85,B 0,C 180,E1 -12883.743,E2 -12883.743} C_VEL
LIN {X 0,Y 371.609,Z 590.122,A -85,B 0,C 180,E1 -12883.886,E2 -12883.886} C_VEL
LIN {X 0,Y 372.905,Z 576.299,A -85,B 0,C 180,E1 -12884.88,E2 -12884.88} C_VEL
LIN {X 0,Y 374.053,Z 562.039,A -85,B 0,C 180,E1 -12885.67,E2 -12885.67} C_VEL
LIN {X 0,Y 374.901,Z 546.685,A -85,B 0,C 180,E1 -12886.297,E2 -12886.297} C_VEL
LIN {X 0,Y 375.516,Z 531.642,A -85,B 0,C 180,E1 -12886.689,E2 -12886.689} C_VEL
LIN {X 0,Y 378.312,Z 410.037,A -85,B 0,C 180,E1 -12889.009,E2 -12889.009} C_VEL
LIN {X 0,Y 372.46,Z 395.135,A -85,B 0,C 180,E1 -12889.767,E2 -12889.767} C_VEL
LIN {X 0,Y 363.069,Z 373.791,A -85,B 0,C 180,E1 -12891.01,E2 -12891.01} C_VEL
LIN {X 0,Y 361.894,Z 369.034,A -85,B 0,C 180,E1 -12892.253,E2 -12892.253} C_VEL
LIN {X 0,Y 361.866,Z 369.033,A -85,B 0,C 180,E1 -12895.295,E2 -12895.295} C_VEL
LIN {X 0,Y 361.859,Z 369.032,A -85,B 0,C 180,E1 -12899.073,E2 -12899.073} C_VEL
LIN {X 0,Y 361.853,Z 369.027,A -85,B 0,C 180,E1 -12902.944,E2 -12902.944} C_VEL
LIN {X 0,Y 361.871,Z 369.027,A -85,B 0,C 180,E1 -12905.637,E2 -12905.637} C_VEL
LIN {X 0,Y 361.829,Z 369.039,A -85,B 0,C 180,E1 -12909.018,E2 -12909.018} C_VEL
LIN {X 0,Y 361.837,Z 369.036,A -85,B 0,C 180,E1 -12912.829,E2 -12912.829} C_VEL
LIN {X 0,Y 361.82,Z 369.025,A -85,B 0,C 180,E1 -12915.947,E2 -12915.947} C_VEL
LIN {X 0,Y 361.816,Z 369.041,A -85,B 0,C 180,E1 -12919.249,E2 -12919.249} C_VEL
LIN {X 0,Y 361.864,Z 369.033,A -85,B 0,C 180,E1 -12922.981,E2 -12922.981} C_VEL
LIN {X 0,Y 361.861,Z 369.029,A -85,B 0,C 180,E1 -12926.631,E2 -12926.631} C_VEL
LIN {X 0,Y 361.859,Z 369.033,A -85,B 0,C 180,E1 -12929.67,E2 -12929.67} C_VEL
LIN {X 0,Y 361.858,Z 368.993,A -85,B 0,C 180,E1 -12933.467,E2 -12933.467} C_VEL
LIN {X 0,Y 361.879,Z 369.021,A -85,B 0,C 180,E1 -12937.143,E2 -12937.143} C_VEL
LIN {X 0,Y 361.89,Z 369.027,A -85,B 0,C 180,E1 -12940.722,E2 -12940.722} C_VEL
LIN {X 0,Y 361.946,Z 369.021,A -85,B 0,C 180,E1 -12944.226,E2 -12944.226} C_VEL
LIN {X 0,Y 362.002,Z 369.012,A -85,B 0,C 180,E1 -12946.527,E2 -12946.527} C_VEL
LIN {X 0,Y 362.002,Z 369.011,A -85,B 0,C 180,E1 -12949.937,E2 -12949.937} C_VEL
LIN {X 0,Y 362.122,Z 368.999,A -85,B 0,C 180,E1 -12953.312,E2 -12953.312} C_VEL
LIN {X 0,Y 362.267,Z 368.986,A -85,B 0,C 180,E1 -12957.776,E2 -12957.776} C_VEL
LIN {X 0,Y 362.178,Z 368.984,A -85,B 0,C 180,E1 -12961.111,E2 -12961.111} C_VEL
LIN {X 0,Y 362.273,Z 368.973,A -85,B 0,C 180,E1 -12962.223,E2 -12962.223} C_VEL
LIN {X 0,Y 362.124,Z 368.996,A -85,B 0,C 180,E1 -12966.687,E2 -12966.687} C_VEL
LIN {X 0,Y 362.002,Z 369.016,A -85,B 0,C 180,E1 -12970.062,E2 -12970.062} C_VEL
LIN {X 0,Y 361.981,Z 369.014,A -85,B 0,C 180,E1 -12973.886,E2 -12973.886} C_VEL
LIN {X 0,Y 361.912,Z 369.02,A -85,B 0,C 180,E1 -12978.101,E2 -12978.101} C_VEL
LIN {X 0,Y 361.891,Z 369.025,A -85,B 0,C 180,E1 -12981.653,E2 -12981.653} C_VEL
LIN {X 0,Y 361.883,Z 369.032,A -85,B 0,C 180,E1 -12985.293,E2 -12985.293} C_VEL
LIN {X 0,Y 361.855,Z 369.034,A -85,B 0,C 180,E1 -12989.073,E2 -12989.073} C_VEL
LIN {X 0,Y 361.849,Z 369.033,A -85,B 0,C 180,E1 -12992.944,E2 -12992.944} C_VEL
LIN {X 0,Y 361.867,Z 369.033,A -85,B 0,C 180,E1 -12995.636,E2 -12995.636} C_VEL
LIN {X 0,Y 361.824,Z 369.03,A -85,B 0,C 180,E1 -12999.017,E2 -12999.017} C_VEL
LIN {X 0,Y 361.832,Z 369.035,A -85,B 0,C 180,E1 -13002.829,E2 -13002.829} C_VEL
LIN {X 0,Y 361.816,Z 369.042,A -85,B 0,C 180,E1 -13005.947,E2 -13005.947} C_VEL
LIN {X 0,Y 361.811,Z 369.041,A -85,B 0,C 180,E1 -13009.249,E2 -13009.249} C_VEL
LIN {X 0,Y 361.862,Z 369.038,A -85,B 0,C 180,E1 -13012.981,E2 -13012.981} C_VEL
LIN {X 0,Y 361.905,Z 369.14,A -85,B 0,C 180,E1 -13014.067,E2 -13014.067} C_VEL
LIN {X 0,Y 365.208,Z 382.262,A -85,B 0,C 180,E1 -13017.068,E2 -13017.068} C_VEL
LIN {X 0,Y 367.774,Z 393.205,A -85,B 0,C 180,E1 -13019.421,E2 -13019.421} C_VEL
LIN {X 0,Y 372.362,Z 405.024,A -85,B 0,C 180,E1 -13020.034,E2 -13020.034} C_VEL
LIN {X 0,Y 377.917,Z 436.171,A -85,B 0,C 180,E1 -13021.103,E2 -13021.103} C_VEL
LIN {X 0,Y 375.049,Z 558.859,A -85,B 0,C 180,E1 -13023.461,E2 -13023.461} C_VEL
LIN {X 0,Y 374.248,Z 573.622,A -85,B 0,C 180,E1 -13023.925,E2 -13023.925} C_VEL
LIN {X 0,Y 373.162,Z 587.228,A -85,B 0,C 180,E1 -13024.532,E2 -13024.532} C_VEL
LIN {X 0,Y 371.993,Z 600.43,A -85,B 0,C 180,E1 -13025.309,E2 -13025.309} C_VEL
LIN {X 0,Y 370.439,Z 614.68,A -85,B 0,C 180,E1 -13026.373,E2 -13026.373} C_VEL
LIN {X 0,Y 368.875,Z 627.852,A -85,B 0,C 180,E1 -13027.601,E2 -13027.601} C_VEL
LIN {X 0,Y 367.19,Z 639.981,A -85,B 0,C 180,E1 -13028.969,E2 -13028.969} C_VEL
LIN {X 0,Y 365.85,Z 650.592,A -85,B 0,C 180,E1 -13030.402,E2 -13030.402} C_VEL
LIN {X 0,Y 364.501,Z 660.733,A -85,B 0,C 180,E1 -13032.031,E2 -13032.031} C_VEL
LIN {X 0,Y 363.088,Z 670.94,A -85,B 0,C 180,E1 -13033.989,E2 -13033.989} C_VEL
LIN {X 0,Y 361.992,Z 679.997,A -85,B 0,C 180,E1 -13036.104,E2 -13036.104} C_VEL
LIN {X 0,Y 361.256,Z 687.342,A -85,B 0,C 180,E1 -13038.213,E2 -13038.213} C_VEL
LIN {X 0,Y 360.706,Z 693.639,A -85,B 0,C 180,E1 -13040.467,E2 -13040.467} C_VEL
LIN {X 0,Y 360.466,Z 698.498,A -85,B 0,C 180,E1 -13042.719,E2 -13042.719} C_VEL
LIN {X 0,Y 360.331,Z 701.305,A -85,B 0,C 180,E1 -13044.403,E2 -13044.403} C_VEL
LIN {X 0,Y 360.287,Z 703.914,A -85,B 0,C 180,E1 -13046.645,E2 -13046.645} C_VEL
LIN {X 0,Y 360.34,Z 705.313,A -85,B 0,C 180,E1 -13048.882,E2 -13048.882} C_VEL
LIN {X 0,Y 360.335,Z 705.563,A -85,B 0,C 180,E1 -13051.118,E2 -13051.118} C_VEL
